# B&R Automation Studio project vibratorControlWithCurrentController
Automation Studio 4.12.5.95 SP; technology packages: Acp10Arnc0 5.23.1

## Configuration CM20

CPU X20CP0484, AutomationRuntime H4.93, Build 4.1.2, Safety 0.0, Vc 

### Task classes (Cpu.sw)
```
Cyclic#1 (cycle 800 us, tolerance 0 us):
  VibratorCo <- modules.main.vibrator.VibratorControl.prg
Cyclic#2 (cycle 1600 us, tolerance 0 us):
  sineWaveGe <- modules.main.vibrator.sineWaveGen.prg [disabled]
  belt <- modules.main.belt.belt.prg
  sampling <- modules.sampling.prg
Cyclic#3 (cycle 4800 us, tolerance 0 us):
  main <- modules.main.main.prg
  feeder <- modules.feeder.feeder.prg
  vibrator <- modules.main.vibrator.vibrator.prg
  EM_vibrat <- modules.main.vibrator.EM_Vibrator.prg
  capcon <- modules.main.capcon.capcon.prg
  wing <- modules.main.wing.wing.prg
  upperFlap <- modules.main.wing.upperFlap.upperFlap.prg
  middleFlap <- modules.main.wing.middleFlap.middleFlap.prg
  bottomFlap <- modules.main.wing.bottomFlap.bottomFlap.prg
  cassette <- modules.main.wing.cassette.cassette.prg
Cyclic#4 (cycle 20000 us, tolerance 1000000 us):
  ethIp <- services.EthernetIP.ethIp.prg
  udpClient <- services.machine.udpClient.prg
  simulation <- simulation.simulation.prg
  lampCtrl <- services.machine.lampCtrl.prg [disabled]
Cyclic#5 (cycle 40000 us, tolerance 1000000 us):
  alarm <- services.alarm.alarm.prg
  file <- services.file.file.prg
  recipe <- services.recipe.recipe.prg
  recipeCurr <- services.recipe.recipeCurrent.prg
  machine <- services.machine.machine.prg
  config <- services.config.config.prg
  updateCM <- services.machine.updateCM.prg
  updateEWU <- services.machine.updateEWU.prg
  elementImg <- services.elementImg.elementImg.prg
  simCapcon <- simulation.capcon.simCapcon.prg [disabled]
  recipeCtrl <- services.recipeCtrl.recipeCtrl.prg
  transferCo <- services.machine.transferConfigToT50.prg
  FAT <- services.FAT.FAT.prg
DataObjects: eipconf <- services.EthernetIP.eipconf.dob, Acp10sys
NcDataObjects: acp10etxen <- acp10etxen.dob, gAxisVibCi <- gAxisVibCobj.gAxisVibCi.dob, cfCurCtr <- gAxisVibCobj.cfCurCtr.dob, gAxisVibLi <- gAxisVibLobj.gAxisVibLi.dob, lfCurCtr <- gAxisVibLobj.lfCurCtr.dob, gAxisBelta <- gAxisBeltobj.gAxisBelta.dob, gAxisBelti <- gAxisBeltobj.gAxisBelti.dob, lfNew <- gAxisVibLobj.lfNew.dob
Binaries: mvLoader, udbdef, FWRules, TCData, TCLang, OpcUaSrv, arsvcreg, acp10cfg, Acp10map, arconfig, User, iomap, asfw, ashwac, ashwd, sysconf, Role, mp_recipe, mp_recipeC, asiol1, User_1, mp_config, mp_data, alarm_hist, TC, mp_user, mp_alarm
Libraries: Acp10man, Acp10par, NcGlobal, VibCtrl, LookupTbl, MpRecipe, MpBase, sys_lib, runtime, MpAlarmX, astime, brdkMC, Acp10_MC, AsBrMath, standard, AsBrStr, brsystem, brdkMU, brdkSIM, brdkCSV, brdkPV, legoCM20, legoSTR, DataObj, brdkOPCUA, AsOpcUas, brdkUpdate, ArProject, brdkFile, AsSem, AsIO, AsOpcUac, FileIO, AsIODiag, AsUSB, brdkREST, brdkJSON, brdkSTR, RandomLib, AsHttp, AsARCfg, AsMath, asstring, AsEthIP, MTFilter, MTTypes, MTBasics, MTLookUp, MTData, MpData, MpServer, Goertzel, EasyUaClnt, AsIOLink, AsIOAcc, AsUDP, powerlnk, arssl, asieccon, aruser, MpReport
```

### Hardware
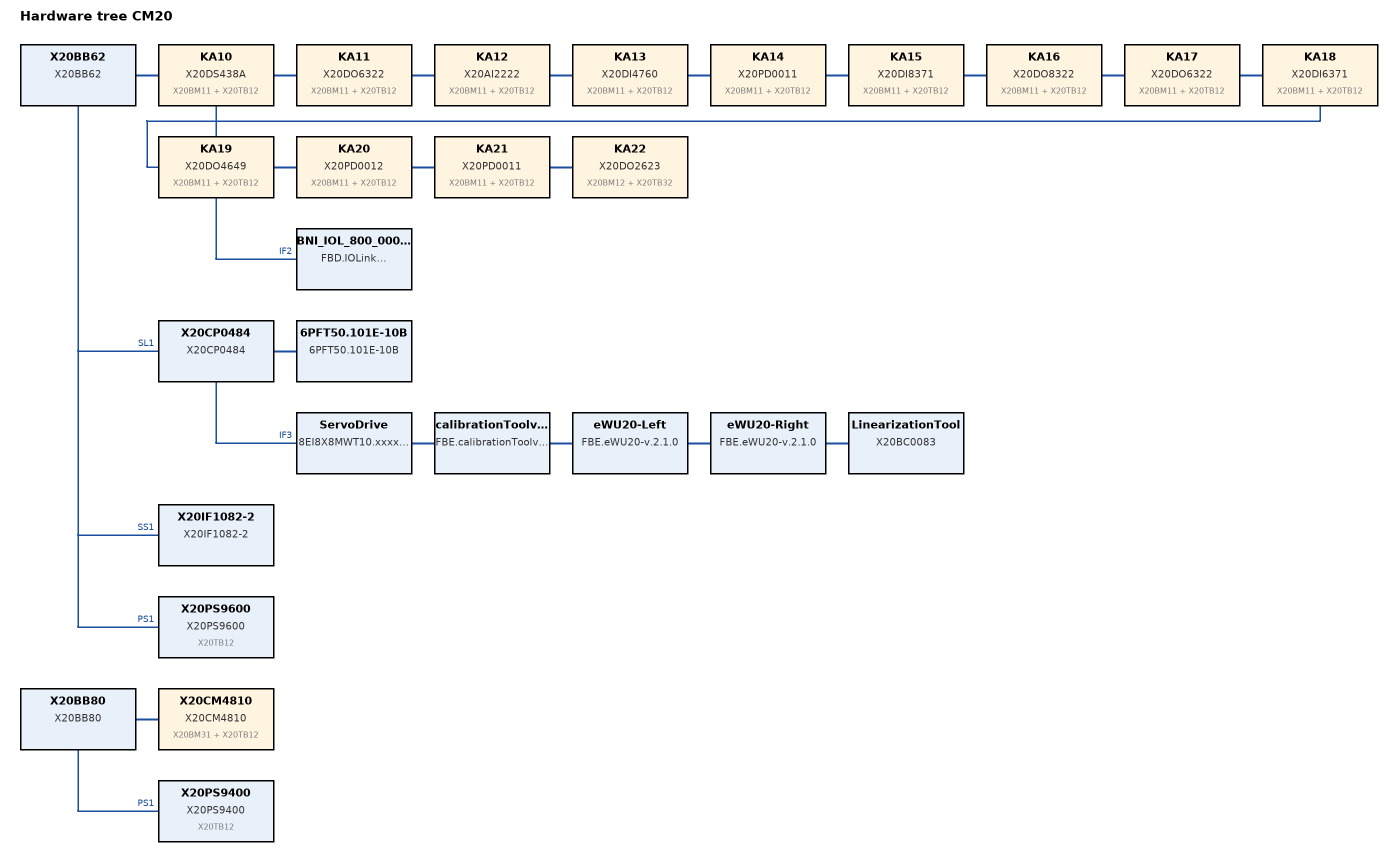
```
6PFT50.101E-10B : 6PFT50.101E-10B v1.4.0.0  [ETH1 -> X20CP0484.IF2 [Cable Type=PowerlinkCable, Length=10, Version=1.0.0.3]]
  Terminal = true
  Startmode = 2
  Mode = Manual
  InternetAddress = 192.168.2.70
  Subnetmask = 255.255.255.0
  ScreenRotation = 270
  PasswordVNC = 
  SelectedFavoriteWeb = 192.168.2.11:81
  USBmemshare = 1
  Usermemshare = 1
  PasswordCIFS = 1234
  UpdateServerType = 2
  UpdateServerFromDhcp = 0
  UpdateServerUser = superuser
  UpdateServerPassword = superuser
  UpdateServerAddress = 192.168.2.11
  PasswordService = 
  ActivateOpcUaServer = 1
BNI_IOL_800_000_Z036_IODD1_1 : FBD.IOLink.GenericDeviceDTM.DTMCore.BNI IOL-800-000-Z036 IODD1.1 v1.8 (OrderNumber=BNI IOL-800-000-Z036 IODD1.1)  [IO-Link1 -> KA10.IF2]
  DtmId = 7a61ab58-0b64-4e0b-ae65-61df76657b3c
KA10 : X20DS438A v2.4.0.0  [SS1 -> X20TB12c.SS; SL -> X20BM11b.SL1]
  DtmRef = FBD.BRIOLinkModuleDTM.DTMCore.X20DS438A
  DtmId = c2005f39-6d59-4b1f-87b2-556bc89c9aff
  CommDtmId = f866141b-695e-453b-bc4e-9ec5edcbb4a9
  RequiresDTMBuild = true
  ConfigFile = Communication.dtm
  ConfigModule = asiol1
  Supervision = off
  OperatingMode01 = DigInput
  OperatingMode02 = Operate
  PDO_Enable02 = variousTypes
  PDO_DataType02_1 = USINT
  OperatingMode03 = DigInput
KA11 : X20DO6322 v1.4.0.0  [SS1 -> X20TB12n.SS; SL -> X20BM11j.SL1]
  Supervision = off
KA12 : X20AI2222 v1.4.0.0  [SS1 -> X20TB12i.SS; SL -> X20BM11h.SL1]
  Supervision = off
KA13 : X20DI4760 v1.2.0.0  [SS1 -> X20TB12p.SS; SL -> X20BM11l.SL1]
  Supervision = off
KA14 : X20PD0011 v1.2.0.0  [SS1 -> X20TB12o.SS; SL -> X20BM11k.SL1]
  Supervision = off
KA15 : X20DI8371 v1.6.0.0  [SS1 -> X20TB12q.SS; SL -> X20BM11m.SL1]
  Supervision = off
KA16 : X20DO8322 v1.8.0.0  [SS1 -> X20TB12r.SS; SL -> X20BM11n.SL1]
  Supervision = off
KA17 : X20DO6322 v1.4.0.0  [SS1 -> X20TB12s.SS; SL -> X20BM11o.SL1]
  Supervision = off
KA18 : X20DI6371 v1.2.0.0  [SS1 -> X20TB12t.SS; SL -> X20BM11p.SL1]
  Supervision = off
KA19 : X20DO4649 v1.2.0.0  [SS1 -> X20TB12u.SS; SL -> X20BM11q.SL1]
  Supervision = off
KA20 : X20PD0012 v1.2.0.0  [SS1 -> X20TB12a.SS; SL -> X20BM11.SL1]
  Supervision = off
KA21 : X20PD0011 v1.2.0.0  [SS1 -> X20TB12b.SS; SL -> X20BM11a.SL1]
  Supervision = off
KA22 : X20DO2623 v1.2.1.0  [SS1 -> X20TB32.SS; SL -> X20BM12.SL1]
  Supervision = off
LinearizationTool : X20BC0083 v2.9.0.0  [PLK1 -> eWU20-Right.PLK2 (NodeNumber=3) [Cable Type=PowerlinkCable, Length=10, Version=1.0.0.3]; SL -> X20BB80.SL1]
  Supervision = off
ServoDrive : 8EI8X8MWT10.xxxx-1 v2.3.2.0  [PLK1 -> X20CP0484.IF3 (NodeNumber=1) [Cable Type=PowerlinkCable, Length=10, Version=1.0.0.3]; PLK2 -> calibrationToolv.1.2.0.PLK1 (NodeNumber=1) [Cable Type=PowerlinkCable, Length=10, Version=1.0.0.3]]
  MotionTP = Acp10Arnc0
  Ax1Interface = Ax1EnDat
X20BB62 : X20BB62 v1.3.0.0
  Connector IF6:
    CycleTime = 1600
    AsyncPayload = 120
    OutputJustInTime = off
X20BB80 : X20BB80 v1.0.2.0
X20BM11 : X20BM11 v1.1.0.0  [X2X1 -> X20BM11q.X2X2]
X20BM11a : X20BM11 v1.1.0.0  [X2X1 -> X20BM11.X2X2]
X20BM11b : X20BM11 v1.1.0.0  [X2X1 -> X20BB62.IF6]
X20BM11h : X20BM11 v1.1.0.0  [X2X1 -> X20BM11j.X2X2]
X20BM11j : X20BM11 v1.1.0.0  [X2X1 -> X20BM11b.X2X2]
X20BM11k : X20BM11 v1.1.0.0  [X2X1 -> X20BM11l.X2X2]
X20BM11l : X20BM11 v1.1.0.0  [X2X1 -> X20BM11h.X2X2]
X20BM11m : X20BM11 v1.1.0.0  [X2X1 -> X20BM11k.X2X2]
X20BM11n : X20BM11 v1.1.0.0  [X2X1 -> X20BM11m.X2X2]
X20BM11o : X20BM11 v1.1.0.0  [X2X1 -> X20BM11n.X2X2]
X20BM11p : X20BM11 v1.1.0.0  [X2X1 -> X20BM11o.X2X2]
X20BM11q : X20BM11 v1.1.0.0  [X2X1 -> X20BM11p.X2X2]
X20BM12 : X20BM12 v1.1.0.0  [X2X1 -> X20BM11a.X2X2]
X20BM31 : X20BM31 v1.1.0.0  [X2X1 -> X20BB80.IF1]
X20CM4810 : X20CM4810 v1.4.4.0  [SS1 -> X20TB12e.SS; SL -> X20BM31.SL1]
  Supervision = off
  AIScale01 = 0x0007
  Current02 = on
  AIScale02 = 0x0060
  AICalc02 = on
  AISamplesSource02 = cyclic
  AIParameter02 = PEAK
X20CP0484 : X20CP0484 v1.7.0.0  [SL -> X20BB62.SL1]
  Connector IF2:
    ActivateDevice = 1
    HostName = countingmachine
    Mode = Manual
    InternetAddress = 192.168.2.11
    SubnetMask = 255.255.255.0
    InaNodeNumber = 0
    ActivateSnmp = 2
  Connector IF3:
    MtuSize = 1500
    CycleTime = 800
    InternetAddress = 192.168.200.240
    SubnetMask = 255.255.255.0
    ActivateANSL = 1
  ConfigurationID = CountingMachine
  ConfigVersion = 2.1.42
  UserPartitionSize = 100
  RemanentGlobalPvSize = 500
  VolatileGlobalPvSize = 455350
  EnableUsbRemoteInstall = 1
  EnableCfRemoteInstall = 1
  TimerDeviceType = EPLX2X
  TimerDevice = X20CP0484.IF3
  IdleTaskClass = 4
  TaskClassIdleTime = 1600
  CyclicTaskClassCount = 5
  Cyclic1Duration = 800
  Cyclic1Tolerance = 0
  Cyclic2Duration = 1600
  Cyclic2Tolerance = 0
  Cyclic3Duration = 4800
  Cyclic3Tolerance = 0
  Cyclic4Duration = 20000
  Cyclic4Tolerance = 1000000
  Cyclic5Duration = 40000
  Cyclic5Tolerance = 1000000
  Cyclic6Duration = 500000
  Cyclic6Tolerance = 500000
  Cyclic7Duration = 1000000
  Cyclic7Tolerance = 1000000
  Cyclic8Duration = 9600
  Cyclic8Tolerance = 30000000
  FileDevice1
  FileDeviceName1 = USER
  FileDevicePath1 = USER_PATH
  TimeZone = 140
  ActivateSntp = 1
  SntpcServAddr1 = 192.168.1.199
  EthernetHostName = cm20
  EthernetDefaultGateway = 192.168.1.254
  ActivateDns = 1
  DnsServer1 = 192.168.1.1
  FtpUser1
  FtpUsername1 = admin
  FtpUserPassword1 = /xeWp7dP4cZARaoRUYb4lC4ZD6ydIPKFJHxZK63t4D4=
  FtpUserSalt1 = z+XtgaLv
  FTPAccessRight1 = 0
  FtpUser2
  FtpUsername2 = superuser
  FtpUserPassword2 = hun78AKmVJbSvtD9VGxdA3Iq+bPiFMAeRRsTULM9hlc=
  FtpUserSalt2 = IDYkuK0C
  FTPAccessRight2 = 0
  FTPdevice2 = ALL
  FtpUser3
  FtpUsername3 = update
  FtpUserPassword3 = +43P0CP5LPvLZS5Hk18lIwvQq9JpaLJM6nsEQnrbHXY=
  FtpUserSalt3 = TaVVG8PK
  FTPAccessRight3 = 0
  FTPMSpath3 = update
  FtpUser4
  FtpUsername4 = updateewu
  FtpUserPassword4 = epKGN9X0JvLfxgCXyMdS0yy+jyVnLXtvgYSXuK2LydA=  // updateewu
  FtpUserSalt4 = ShQX0Ew+
  FTPAccessRight4 = 0
  FTPMSpath4 = updateewu
  ActivateOpcUa = 1
  OpcUaInformationModels_PV_Version = 2
  OpcUaInformationModel_Facet = 0
  OpcUaInformationModel_TypeInformation = 0
  OpcUaInformationModel_BaseObjectTypeForStructures = 0
X20IF1082-2 : X20IF1082-2 v1.15.0.0  [SS -> X20BB62.SS1]
  Connector IF1:
    Operation = EthOnly
    HostName = cm20
    ActivateANSL = 1
    ActivateSnmp = 2
X20PS9400 : X20PS9400 v1.8.0.0  [SS1 -> X20TB12d.SS; PS -> X20BB80.PS1]
  Supervision = off
X20PS9600 : X20PS9600 v1.6.1.0  [PS -> X20BB62.PS1; SS1 -> X20TB12.SS]
X20TB12 : X20TB12 v1.0.0.0
X20TB12a : X20TB12 v1.0.0.0
X20TB12b : X20TB12 v1.0.0.0
X20TB12c : X20TB12 v1.0.0.0
X20TB12d : X20TB12 v1.0.0.0
X20TB12e : X20TB12 v1.0.0.0
X20TB12i : X20TB12 v1.0.0.0
X20TB12n : X20TB12 v1.0.0.0
X20TB12o : X20TB12 v1.0.0.0
X20TB12p : X20TB12 v1.0.0.0
X20TB12q : X20TB12 v1.0.0.0
X20TB12r : X20TB12 v1.0.0.0
X20TB12s : X20TB12 v1.0.0.0
X20TB12t : X20TB12 v1.0.0.0
X20TB12u : X20TB12 v1.0.0.0
X20TB32 : X20TB32 v1.0.0.1
calibrationToolv.1.2.0 : FBE.calibrationToolv.1.2.0 v1.0 (OrderNumber=calibrationToolv.1.2.0)  [PLK1 -> ServoDrive.PLK2 (NodeNumber=2) [Cable Type=PowerlinkCable, Length=10, Version=1.0.0.3]; PLK2 -> eWU20-Left.PLK1 (NodeNumber=2) [Cable Type=PowerlinkCable, Length=10, Version=1.0.0.3]]
  Supervision = off
  pA240s01_direction = ro
  pA240s03_direction = ro
  pA500s01_direction = wo
eWU20-Left : FBE.eWU20-v.2.1.0 v1.0 (OrderNumber=eWU20-Left)  [PLK1 -> calibrationToolv.1.2.0.PLK2 (NodeNumber=20) [Cable Type=PowerlinkCable, Length=10, Version=1.0.0.3]; PLK2 -> eWU20-Right.PLK1 (NodeNumber=20) [Cable Type=PowerlinkCable, Length=10, Version=1.0.0.3]]
  Supervision = off
  pA080s01_direction = ro
  pA080s02_direction = ro
  pA080s03_direction = ro
  pA080s04_direction = ro
  pA080s05_direction = ro
  pA080s06_direction = ro
  pA080s07_direction = ro
  pA080s08_direction = ro
  pA080s09_direction = ro
  pA080s0A_direction = ro
  pA080s0B_direction = ro
  pA500s01_direction = wo
  pA500s02_direction = wo
  pA500s03_direction = wo
  pA500s04_direction = wo
  pA500s05_direction = wo
  pA500s06_direction = wo
  pA500s07_direction = wo
  pA500s08_direction = wo
  pA500s09_direction = wo
  pA500s0A_direction = wo
  pA500s0B_direction = wo
  pA500s0C_direction = wo
  pA500s0D_direction = wo
  pA500s0E_direction = wo
  pA1C0s01_direction = ro
  pA1C0s02_direction = ro
  pA1C0s03_direction = ro
  pA1C0s04_direction = ro
eWU20-Right : FBE.eWU20-v.2.1.0 v1.0 (OrderNumber=eWU20-Left)  [PLK1 -> eWU20-Left.PLK2 (NodeNumber=21) [Cable Type=PowerlinkCable, Length=10, Version=1.0.0.3]; PLK2 -> LinearizationTool.PLK1 (NodeNumber=21) [Cable Type=PowerlinkCable, Length=10, Version=1.0.0.3]]
  Supervision = off
  pA080s01_direction = ro
  pA080s02_direction = ro
  pA080s03_direction = ro
  pA080s04_direction = ro
  pA080s05_direction = ro
  pA080s06_direction = ro
  pA080s07_direction = ro
  pA080s08_direction = ro
  pA080s09_direction = ro
  pA080s0A_direction = ro
  pA080s0B_direction = ro
  pA500s01_direction = wo
  pA500s02_direction = wo
  pA500s03_direction = wo
  pA500s04_direction = wo
  pA500s05_direction = wo
  pA500s06_direction = wo
  pA500s07_direction = wo
  pA500s08_direction = wo
  pA500s09_direction = wo
  pA500s0A_direction = wo
  pA500s0B_direction = wo
  pA500s0C_direction = wo
  pA500s0D_direction = wo
  pA500s0E_direction = wo
  pA1C0s01_direction = ro
  pA1C0s02_direction = ro
  pA1C0s03_direction = ro
  pA1C0s04_direction = ro
```

### Cpu.pkg.orig - X20CP0484/Cpu.pkg.orig
(orig body not rendered)

### IoMap.iom - X20CP0484/IoMap.iom
```iecst
VAR_CONFIG
	::feeder:this.hw.do_levelSensorInBowlLow AT %QX."KA11".DigitalOutput01;
	::feeder:this.hw.do_levelSensorInBowlMedium AT %QX."KA11".DigitalOutput03;
	::feeder:this.hw.do_levelSensorInBowlHigh AT %QX."KA11".DigitalOutput05;
	::main:this.hw.do_alarmBeacon AT %QX."KA11".DigitalOutput02;
	::main:this.alarm.KA11.active AT %IX."KA11".ModuleOk;
	::feeder:this.hw.do_beltForwards AT %QX."KA11".DigitalOutput04;
	::feeder:this.hw.do_beltBackwards AT %QX."KA11".DigitalOutput06;
	::main:this.alarm.KA12.active AT %IX."KA12".ModuleOk;
	::sampling:this.hw.ai_signal[1] AT %IW."KA12".AnalogInput01;
	::sampling:this.hw.di_upperFlap_change AT %IX."KA13".DigitalInput01;
	::sampling:this.hw.di_bottomFlap_change AT %IX."KA13".DigitalInput02;
	::sampling:this.hw.di_middleFlap_change AT %IX."KA13".DigitalInput03;
	::sampling:this.hw.di_neigbourFlap_change AT %IX."KA13".DigitalInput04;
	::main:this.alarm.KA14.active AT %IX."KA13".ModuleOk;
	::main:this.alarm.KA13.active AT %IX."KA14".ModuleOk;
	::cassette:this.hwAir.di_neighbourActive AT %IX."KA15".DigitalInput02;
	::cassette:this.hwAir.di_cassetteReady AT %IX."KA15".DigitalInput03;
	::bottomFlap:this.hwAir.di_neighbourPortionReady AT %IX."KA15".DigitalInput05;
	::cassette:this.hwAir.di_cassetteQueue AT %IX."KA15".DigitalInput01;
	::bottomFlap:this.hwAir.di_neighbourActive AT %IX."KA15".DigitalInput02;
	::cassette:this.hwAir.di_neighbourIsDosing AT %IX."KA15".DigitalInput04;
	::cassette:this.hwAir.di_neighbourBricksInCassette AT %IX."KA15".DigitalInput07;
	::main:this.alarm.KA15.active AT %IX."KA15".ModuleOk;
	::bottomFlap:this.hwAir.di_neigbourIsDosing AT %IX."KA15".DigitalInput04;
	::upperFlap:this.hw.do_open AT %QX."KA16".DigitalOutput01;
	::middleFlap:this.hw.do_open AT %QX."KA16".DigitalOutput03;
	::bottomFlap:this.hw.do_neighbourPortionReady AT %QX."KA16".DigitalOutput05;
	::cassette:this.hw.do_bricksReadyInCassette AT %QX."KA16".DigitalOutput07;
	::cassette:this.hw.do_dosing AT %QX."KA16".DigitalOutput04;
	::wing:this.hw.do_active AT %QX."KA16".DigitalOutput02;
	::main:this.alarm.KA16.active AT %IX."KA16".ModuleOk;
	::feeder:this.hw.do_beltForwards AT %QX."KA16".DigitalOutput06;
	::feeder:this.hw.do_beltBackwards AT %QX."KA16".DigitalOutput08;
	::bottomFlap:this.hw.do_open AT %QX."KA17".DigitalOutput01;
	::bottomFlap:this.hw.do_neighbourOpen AT %QX."KA17".DigitalOutput03;
	::cassette:this.hw.do_cassetteRelease AT %QX."KA17".DigitalOutput05;
	::main:this.alarm.KA17.active AT %IX."KA17".ModuleOk;
	::feeder:this.hw.di_flapIsClosed AT %IX."KA18".DigitalInput02;
	::feeder:this.hw.di_levelSensorBelt AT %IX."KA18".DigitalInput03;
	::feeder:this.hw.di_flapIsOpen AT %IX."KA18".DigitalInput04;
	::feeder:this.hw.di_boxIsReadyAtFlap AT %IX."KA18".DigitalInput05;
	::main:this.alarm.KA18.active AT %IX."KA18".ModuleOk;
	::feeder:this.hw.do_flapClose AT %QX."KA19".DigitalOutput01;
	::feeder:this.hw.do_flapClose AT %QX."KA19".DigitalOutput04;
	::feeder:this.hw.do_flapOpen AT %QX."KA19".DigitalOutput02;
	::feeder:this.hw.do_flapOpen AT %QX."KA19".DigitalOutput03;
	::main:this.alarm.KA19.active AT %IX."KA19".ModuleOk;
	::main:this.alarm.KA20.active AT %IX."KA20".ModuleOk;
	::main:this.alarm.KA21.active AT %IX."KA21".ModuleOk;
	::main:this.alarm.KA10.active AT %IX."KA10".ModuleOk;
	::feeder:this.hw.di_levelSensorInBowl AT %IX."KA10".DigitalInput01;
	::belt:this.hw.di_photo AT %IX."KA10".DigitalInput03;
	::VibratorCo:localVariables[1].Accelerometer_0.ai_peakValue AT %ID."calibrationToolv.1.2.0".AnalogValue_IA240_S01;
	::VibratorCo:localVariables[1].Accelerometer_0.ai_rawValue AT %ID."calibrationToolv.1.2.0".RawVib_IA240_S03;
	::VibratorCo:localVariables[0].Accelerometer_0.ai_rawValue AT %ID."calibrationToolv.1.2.0".RawVib_IA240_S03;
	::sineWaveGe:acc.analogVib AT %ID."calibrationToolv.1.2.0".AnalogValue_IA240_S01;
	::VibratorCo:localVariables[0].Accelerometer_0.ai_peakValue AT %ID."calibrationToolv.1.2.0".AnalogValue_IA240_S01;
	::EM_vibrat:localVariables[0].hw.ModuleOkCalibrationTool AT %IX."calibrationToolv.1.2.0".ModuleOk;
	::EM_vibrat:localVariables[1].hw.ModuleOkCalibrationTool AT %IX."calibrationToolv.1.2.0".ModuleOk;
	::VibratorCo:localVariables[0].Accelerometer_0.ModuleOkCalibrationTool AT %IX."calibrationToolv.1.2.0".ModuleOk;
	::VibratorCo:localVariables[1].Accelerometer_0.ModuleOkCalibrationTool AT %IX."calibrationToolv.1.2.0".ModuleOk;
	::cassette:this.hwWu[1].di_wingUnitActive AT %IX."eWU20-Right".WuConnected_IA080_S01;
	::bottomFlap:this.hwWu[1].neighbourActive AT %IX."eWU20-Right".StatusNeighbourActive_IA080_S02;
	::cassette:this.hwWu[0].di_wingUnitActive AT %IX."eWU20-Left".WuConnected_IA080_S01;
	::upperFlap:this.hwWu[0].di_wingUnitActive AT %IX."eWU20-Left".WuConnected_IA080_S01;
	::middleFlap:this.hwWu[0].di_wingUnitActive AT %IX."eWU20-Left".WuConnected_IA080_S01;
	::bottomFlap:this.hwWu[0].di_wingUnitActive AT %IX."eWU20-Left".WuConnected_IA080_S01;
	::bottomFlap:this.hwWu[0].neighbourActive AT %IX."eWU20-Left".StatusNeighbourActive_IA080_S02;
	::bottomFlap:this.hwWu[0].neigbourIsDosing AT %IX."eWU20-Left".Di_bottomFlap_neighbourIsDosing_IA080_S03;
	::bottomFlap:this.hwWu[0].neighbourPortionReady AT %IX."eWU20-Left".Di_bottomFlap_neighbourPortReady_IA080_S04;
	::cassette:this.hwWu[0].di_cassetteQueue AT %IX."eWU20-Left".Di_cassette_queue_IA080_S05;
	::cassette:this.hwWu[0].di_neighbourActive AT %IX."eWU20-Left".Di_cassette_neighbourActive_IA080_S06;
	::cassette:this.hwWu[0].di_cassetteReady AT %IX."eWU20-Left".Di_cassette_ready_IA080_S07;
	::cassette:this.hwWu[0].di_neighbourIsDosing AT %IX."eWU20-Left".Di_cassette_neighbourIsDosing_IA080_S08;
	::cassette:this.hwWu[0].di_neighbourBricksInCassette AT %IX."eWU20-Left".Di_cassette_neighbourBricksInCas_IA080_S09;
	::bottomFlap:cm20Connected AT %QX."eWU20-Left".CM20connected_IA500_S01;
	::upperFlap:this.flap.do_open AT %QX."eWU20-Left".Do_upperFlap_open_IA500_S02;
	::middleFlap:this.flap.do_open AT %QX."eWU20-Left".Do_middleFlap_open_IA500_S03;
	::bottomFlap:this.flap.do_open AT %QX."eWU20-Left".Do_bottomFlap_open_IA500_S04;
	::bottomFlap:this.hw.do_neighbourPortionReady AT %QX."eWU20-Left".Do_bottomFlap_neighbourPortReady_IA500_S06;
	::bottomFlap:this.neighbourFlap.do_open AT %QX."eWU20-Left".Do_bottomFlap_neighbourOpen_IA500_S07;
	::cassette:this.hwWu[0].do_active AT %QX."eWU20-Left".Do_cm_active_IA500_S09;
	::cassette:this.hw.do_bricksReadyInCassette AT %QX."eWU20-Left".Do_cassette_BricksReadyInCasette_IA500_S0A;
	::cassette:this.hw.do_cassetteRelease AT %QX."eWU20-Left".Do_cassette_cassetteRelease_IA500_S0B;
	::upperFlap:this.hwWu[0].flapPosition AT %ID."eWU20-Left".Di_upperFlap_positionStatus_IA1C0_S01;
	::middleFlap:this.hwWu[0].flapPosition AT %ID."eWU20-Left".Di_middleFlap_positionStatus_IA1C0_S02;
	::bottomFlap:this.hwWu[0].flapPosition AT %ID."eWU20-Left".Di_bottomFlap_positionStatus_IA1C0_S03;
	::bottomFlap:this.hwWu[0].neighbourFlapPosition AT %ID."eWU20-Left".Di_neighbourFlap_positionStatus_IA1C0_S04;
	::upperFlap:this.hwWu[1].di_wingUnitActive AT %IX."eWU20-Right".WuConnected_IA080_S01;
	::middleFlap:this.hwWu[1].di_wingUnitActive AT %IX."eWU20-Right".WuConnected_IA080_S01;
	::bottomFlap:this.hwWu[1].di_wingUnitActive AT %IX."eWU20-Right".WuConnected_IA080_S01;
	::bottomFlap:this.hwWu[1].neigbourIsDosing AT %IX."eWU20-Right".Di_bottomFlap_neighbourIsDosing_IA080_S03;
	::bottomFlap:this.hwWu[1].neighbourPortionReady AT %IX."eWU20-Right".Di_bottomFlap_neighbourPortReady_IA080_S04;
	::cassette:this.hwWu[1].di_cassetteQueue AT %IX."eWU20-Right".Di_cassette_queue_IA080_S05;
	::cassette:this.hwWu[1].di_neighbourActive AT %IX."eWU20-Right".Di_cassette_neighbourActive_IA080_S06;
	::cassette:this.hwWu[1].di_cassetteReady AT %IX."eWU20-Right".Di_cassette_ready_IA080_S07;
	::cassette:this.hwWu[1].di_neighbourIsDosing AT %IX."eWU20-Right".Di_cassette_neighbourIsDosing_IA080_S08;
	::cassette:this.hwWu[1].di_neighbourBricksInCassette AT %IX."eWU20-Right".Di_cassette_neighbourBricksInCas_IA080_S09;
	::bottomFlap:cm20Connected AT %QX."eWU20-Right".CM20connected_IA500_S01;
	::upperFlap:this.flap.do_open AT %QX."eWU20-Right".Do_upperFlap_open_IA500_S02;
	::middleFlap:this.flap.do_open AT %QX."eWU20-Right".Do_middleFlap_open_IA500_S03;
	::bottomFlap:this.flap.do_open AT %QX."eWU20-Right".Do_bottomFlap_open_IA500_S04;
	::bottomFlap:this.hw.do_neighbourPortionReady AT %QX."eWU20-Right".Do_bottomFlap_neighbourPortReady_IA500_S06;
	::bottomFlap:this.neighbourFlap.do_open AT %QX."eWU20-Right".Do_bottomFlap_neighbourOpen_IA500_S07;
	::cassette:this.hwWu[1].do_active AT %QX."eWU20-Right".Do_cm_active_IA500_S09;
	::cassette:this.hw.do_bricksReadyInCassette AT %QX."eWU20-Right".Do_cassette_BricksReadyInCasette_IA500_S0A;
	::cassette:this.hw.do_cassetteRelease AT %QX."eWU20-Right".Do_cassette_cassetteRelease_IA500_S0B;
	::upperFlap:this.hwWu[1].flapPosition AT %ID."eWU20-Right".Di_upperFlap_positionStatus_IA1C0_S01;
	::middleFlap:this.hwWu[1].flapPosition AT %ID."eWU20-Right".Di_middleFlap_positionStatus_IA1C0_S02;
	::bottomFlap:this.hwWu[1].flapPosition AT %ID."eWU20-Right".Di_bottomFlap_positionStatus_IA1C0_S03;
	::bottomFlap:this.hwWu[1].neighbourFlapPosition AT %ID."eWU20-Right".Di_neighbourFlap_positionStatus_IA1C0_S04;
	::wing:this.hw.wu_error[0] AT %IX."eWU20-Left".Wu_error_IA080_S0A;
	::wing:this.hw.wu_error[1] AT %IX."eWU20-Right".Wu_error_IA080_S0A;
	::main:this.hw.do_wo_ON AT %QX."eWU20-Left".Di_CMRunning_IA500_S0C;
	::main:this.hw.do_wo_ON AT %QX."eWU20-Right".Di_CMRunning_IA500_S0C;
	::main:this.hw.do_clearWU AT %QX."eWU20-Left".Do_clearWU_IA500_S0D;
	::main:this.hw.do_clearWU AT %QX."eWU20-Right".Do_clearWU_IA500_S0D;
	::machine:this.warmRestartWU AT %QX."eWU20-Left".Do_warmRestartWU_IA500_S0E;
	::machine:this.warmRestartWU AT %QX."eWU20-Right".Do_warmRestartWU_IA500_S0E;
	::cassette:this.hw.do_dosing AT %QX."eWU20-Left".Do_bottomFlap_dosing_IA500_S05;
	::cassette:this.hw.do_dosing AT %QX."eWU20-Right".Do_bottomFlap_dosing_IA500_S05;
	::main:this.hw.di_stepperWUExecute[0] AT %IX."eWU20-Left".Di_WU_execute_IA080_S0B;
	::main:this.hw.di_stepperWUExecute[1] AT %IX."eWU20-Right".Di_WU_execute_IA080_S0B;
	::main:this.hw.output_lightTowerBalluff AT %QB."KA10".OutputData02_1;
	::VibratorCo:localVariables[0].Accelerometer_0.isBigCF AT %QX."calibrationToolv.1.2.0".IsBigCF_IA500_S01;
	::VibratorCo:localVariables[1].Accelerometer_0.ai_peakValueBusCtrl AT %ID."X20CM4810".AnalogInput02;
	Cyclic#1.::VibratorCo:localVariables[0].Accelerometer_0.ai_peakValueBusCtrl AT %ID."X20CM4810".AnalogInput02;
	::VibratorCo:localVariables[0].Accelerometer_0.do_enableSampling AT %QX."X20CM4810".AnalogInputControl02;
	::VibratorCo:localVariables[0].Accelerometer_0.ao_samples AT %QW."X20CM4810".AnalogInputSamples02;
	::VibratorCo:localVariables[1].Accelerometer_0.ai_rawValueBusCtrl AT %ID."X20CM4810".AnalogInput01;
	::VibratorCo:localVariables[0].Accelerometer_0.ai_rawValueBusCtrl AT %ID."X20CM4810".AnalogInput01;
	::VibratorCo:localVariables[0].Accelerometer_0.ModuleOkBusCtrl AT %IX."X20CM4810".ModuleOk;
	::VibratorCo:localVariables[1].Accelerometer_0.ModuleOkBusCtrl AT %IX."X20CM4810".ModuleOk;
	::EM_vibrat:localVariables[1].hw.ModuleOkCalibrationToolBusCtrl AT %IX."X20CM4810".ModuleOk;
	::EM_vibrat:localVariables[0].hw.ModuleOkCalibrationToolBusCtrl AT %IX."X20CM4810".ModuleOk;
	::main:this.hw.input_lightTowerBalluff AT %IB."KA10".ChannelStatus02;
END_VAR
```

### Acp10cfg.ncc - X20CP0484/Motion/Acp10cfg.ncc
```
NcConfiguration (Version=5.12.2, NcSwId=Acp10)
  ACP10CF1_typ:
    cnt_nettrc_rec_drive = 1500
    bufsize_trace_upload = 1200
    tc_nc_man_task = Cyclic #2
    glob_pv_as_ncobject = Yes
    ncsys_dl_broadcast = Yes
    ncsys_dl_acp_reset = Yes
    safemc_log_err_to_ax = Yes
    network_init:
      ncsw_init_execute = Yes
      automatic_execute = Yes
      node_nr_warning = Yes
      net_err_before_ncact = Yes
    nettrc:
      enter_parsecrec = Yes
      enter_ncaction = Yes
      save_ring_startidx = Yes
    cam_prof_download:
      cam_dat_dl_parallel = No
      tc_cam_dl_parallel = Task class for NC Manager task
    plk_if[0]:
      if_name = IF3
      tc_CycDat_PLCopen = Cyclic #1
      mc_broadcast_extdat = No
    plk_if[1]:
      if_name = IF1
      tc_CycDat_PLCopen = Task class for NC Manager task
      mc_broadcast_extdat = No
```

### Acp10map.ncm - X20CP0484/Motion/Acp10map.ncm
```
NcMapping (NcSwId=Acp10, DisabledNodesAreHidden=False)
  NcObject gAxisBelt (ModuleId=ServoDrive, Type=ncAXIS, Channel=1, AcoposSimulation=Off, InitParameter=gAxisBelti, AcoposParameter=gAxisBelta, Disabled=FALSE, ModuleDisabled=FALSE)
  NcObject gAxisVibL (ModuleId=ServoDrive, Type=ncAXIS, Channel=2, AcoposSimulation=Off, InitParameter=gAxisVibLi, AcoposParameter=lfNew, Disabled=FALSE, ModuleDisabled=FALSE)
  NcObject 8EI8X8MWT10.xxxx-1_ncV_AXIS1 (ModuleId=ServoDrive, Type=ncV_AXIS, Channel=1, Disabled=TRUE, ModuleDisabled=FALSE)
  NcObject 8EI8X8MWT10.xxxx-1_ncV_AXIS2 (ModuleId=ServoDrive, Type=ncV_AXIS, Channel=2, Disabled=TRUE, ModuleDisabled=FALSE)
  NcObject gAxisVibC (ModuleId=ServoDrive, Type=ncAXIS, Channel=3, AcoposSimulation=Off, InitParameter=gAxisVibCi, AcoposParameter=cfCurCtr, Disabled=FALSE, ModuleDisabled=FALSE)
  NcObject ServoDrive_ncV_AXIS3 (ModuleId=ServoDrive, Type=ncV_AXIS, Channel=3, AcoposSimulation=off, Disabled=true, ModuleDisabled=FALSE)
```

### beltCapcon.vvm - X20CP0484/beltCapcon.vvm
```iecst
(*Belt --> Capcon*)
(*Capcon --> Belt*)
VAR_CONFIG
	Cyclic#3.gCapconInterface.status.ready AT %Q.Cyclic#2.gBeltInterface.cmd.dropBrick; (*Command to belt that the capcon is ready for a brick*)
	Cyclic#3.::gCapconInterface.status.numBricksInPortion AT %Q.Cyclic#2.::gBeltInterface.parameter.brickCountInPortion; (*Insert your comment here...*)
END_VAR
```

### beltFeeder.vvm - X20CP0484/beltFeeder.vvm
```iecst
(*Belt --> Feeder*)
VAR_CONFIG
	Cyclic#2.::gBeltInterface.status.speed AT %Q.Cyclic#3.::gFeederInterface.cmd.speed; (*Insert your comment here...*)
END_VAR
```

### capconWing.vvm - X20CP0484/capconWing.vvm
```iecst
VAR_CONFIG
	Cyclic#3.gWingInterface.status.request AT %Q.Cyclic#3.gCapconInterface.cmd.wingRequest; (*Insert your comment here...*)
	Cyclic#3.gWingInterface.status.ready AT %Q.Cyclic#3.gCapconInterface.cmd.wingReady; (*Insert your comment here...*)
	Cyclic#3.::gCapconInterface.status.wingStartBrickNOK AT %Q.Cyclic#3.::gWingInterface.cmd.startBrickNOK; (*Start wing with brick NOK.*)
	Cyclic#3.::gCapconInterface.status.wingStartBrickOK AT %Q.Cyclic#3.::gWingInterface.cmd.startBrickOK; (*Start wing with brick OK.*)
	Cyclic#3.::gCapconInterface.status.wingStart AT %Q.Cyclic#3.::gWingInterface.cmd.startBrick; (*Start wing without status yet*)
	Cyclic#3.::gWingInterface.status.commandAck AT %Q.Cyclic#3.gCapconInterface.cmd.wingCmdAck; (*Insert your comment here...*)
	Cyclic#3.::gCapconInterface.status.wingDosing AT %Q.Cyclic#3.::gCassetteInterface.cmd.dosing; (*Insert your comment here...*)
END_VAR
```

### mainBelt.vvm - X20CP0484/mainBelt.vvm
```iecst
(*Main --> Belt*)
VAR_CONFIG
	Cyclic#3.::gMainInterface.status.doCalibrate AT %Q.Cyclic#3.::gBeltInterface.cmd.calibrate; (*Insert your comment here...*)
END_VAR
(*Belt --> Main*)
VAR_CONFIG
	Cyclic#3.::gBeltInterface.status.calibratingMode AT %Q.Cyclic#3.::gMainInterface.cmd.activateCalibrateMode[0]; (*Insert your comment here...*)
END_VAR
```

### mainCapcon.vvm - X20CP0484/mainCapcon.vvm
```iecst
(*Main --> Capcon*)
VAR_CONFIG
	Cyclic#3.::gMainInterface.status.doCalibrate AT %Q.Cyclic#3.::gCapconInterface.cmd.emptyStop; (*Insert your comment here...*)
	Cyclic#3.::gMainInterface.status.emptying AT %Q.Cyclic#3.::gCapconInterface.cmd.skipTeach; (*Insert your comment here...*)
END_VAR
(*Capon --> Main*)
VAR_CONFIG
	Cyclic#3.gCapconInterface.status.waiting AT %Q.Cyclic#3.::gMainInterface.cmd.capconWaiting; (*Command to belt that the capcon is ready for a brick*)
END_VAR
```

### mainFeeder.vvm - X20CP0484/mainFeeder.vvm
```iecst
(*Main --> Feeder*)
VAR_CONFIG
	Cyclic#3.::gMainInterface.status.feederStart AT %Q.Cyclic#3.::gFeederInterface.cmd.start; (*Insert your comment here...*)
	Cyclic#3.::gMainInterface.status.feederStop AT %Q.Cyclic#3.::gFeederInterface.cmd.stop; (*Insert your comment here...*)
END_VAR
```

### mainToWing.vvm - X20CP0484/mainToWing.vvm
```iecst
(*Main --> Wing*)
VAR_CONFIG
	Cyclic#3.::gMainInterface.line.emptyMode AT %Q.Cyclic#3.::gWingInterface.cmd.shaftModeEmpty; (*Insert your comment here...*)
	Cyclic#3.::gBottomFlapInterface.status.ready1 AT %Q.Cyclic#3.::gMainInterface.cmd.wingReadyToEmpty; (*Insert your comment here...*)
END_VAR
```

### mainVibr.vvm - X20CP0484/mainVibr.vvm
```iecst
(*Main --> vibrators*)
VAR_CONFIG
	Cyclic#3.::gMainInterface.status.doCalibrate AT %Q.Cyclic#3.::gVibratorInterface[0].cmd.calibrate; (*Insert your comment here...*)
	Cyclic#3.::gMainInterface.status.doCalibrate AT %Q.Cyclic#3.::gVibratorInterface[1].cmd.calibrate; (*Insert your comment here...*)
END_VAR
(*Vibrators --> main*)
VAR_CONFIG
	Cyclic#3.::gVibratorInterface[1].status.calibratingMode AT %Q.Cyclic#3.::gMainInterface.cmd.activateCalibrateMode[2]; (*Insert your comment here...*)
	Cyclic#3.::gVibratorInterface[0].status.calibratingMode AT %Q.Cyclic#3.::gMainInterface.cmd.activateCalibrateMode[1]; (*Insert your comment here...*)
END_VAR
```

### alarm_hist.mpalarmxhistory - X20CP0484/mappServices/alarm_hist.mpalarmxhistory
```
Element mpAlarmXHistory (Type=mpalarmxhistory)
```

### mp_alarm.mpalarmxcore - X20CP0484/mappServices/mp_alarm.mpalarmxcore
```
Element mpAlarmXCore (Type=mpalarmxcore)
  mapp.AlarmX.Core:
    BySeverity:
      [0]:
        Severity = 1  // severity 1 abort Main
        [0] = Reaction
          Name = abortMain
        [1] = Reaction
          Name = alarmBeaconFlash
      [1]:
        Severity = 10  // Severity 10 is abort  Feeder
        [0] = Reaction
          Name = alarmBeaconFlash
        [1] = Reaction
          Name = abortFeeder
      [2]:
        Severity = 20  // Severity 20 is abort CF
        [0] = Reaction
          Name = abortMain
        [1] = Reaction
          Name = alarmBeaconFlash
        [2] = Reaction
          Name = abortCircularFeeder
      [3]:
        Severity = 30  // Severity 30 is abort LF
        [0] = Reaction
          Name = abortMain
        [1] = Reaction
          Name = alarmBeaconFlash
        [2] = Reaction
          Name = abortLinearFeeder
      [4]:
        Severity = 40  // Severity 40 is abort Belt
        [0] = Reaction
          Name = abortMain
        [1] = Reaction
          Name = alarmBeaconFlash
        [2] = Reaction
          Name = abortBelt
      [5]:
        Severity = 50  // Severity 50 is abort Capcon
        [0] = Reaction
          Name = abortMain
        [1] = Reaction
          Name = alarmBeaconFlash
        [2] = Reaction
          Name = abortCapcon
      [6]:
        Severity = 60  // Severity 60 is abort Wing
        [0] = Reaction
          Name = abortWing
        [1] = Reaction
          Name = alarmBeaconFlash
        [2] = Reaction
          Name = abortMain
      [7]:
        Severity = 70
        [0] = Reaction
          Name = abortMain
        [1] = Reaction
          Name = abortFeeder
      [8]:
        Severity = 1000  // Severity 1000 is a warning - will show constant light on alarm beacon
        [0] = Reaction
          Name = alarmBeaconOn
      [9]:
        Severity = 1001  // Severity 1001 is a warning - will blink the alarm beacon slow.
        [0] = Reaction
          Name = alarmBeaconFlashSlow
  mapp.AlarmX.Core.Configuration:
    [0]:
      Name = KA10ModuleError
      Message = {$MainAlarms/KA10ModuleError}
      Code = 100
    [1]:
      Name = KA11ModuleError
      Message = {$MainAlarms/KA11ModuleError}
      Code = 101
    [2]:
      Name = KA12ModuleError
      Message = {$MainAlarms/KA12ModuleError}
      Code = 102
    [3]:
      Name = KA13ModuleError
      Message = {$MainAlarms/KA13ModuleError}
      Code = 103
    [4]:
      Name = KA14ModuleError
      Message = {$MainAlarms/KA14ModuleError}
      Code = 104
    [5]:
      Name = KA15ModuleError
      Message = {$MainAlarms/KA15ModuleError
      Code = 105
    [6]:
      Name = KA16ModuleError
      Message = {$MainAlarms/KA16ModuleError}
      Code = 106
    [7]:
      Name = KA17ModuleError
      Message = {$MainAlarms/KA17ModuleError}
      Code = 107
    [8]:
      Name = KA18ModuleError
      Message = {$MainAlarms/KA18ModuleError}
      Code = 108
    [9]:
      Name = KA19ModuleError
      Message = {$MainAlarms/KA19ModuleError}
      Code = 109
    [10]:
      Name = KA20ModuleError
      Message = {$MainAlarms/KA20ModuleErrorr}
      Code = 110
    [11]:
      Name = feederLowLevel
      Message = {$FeederAlarms/lowLevel}
      Code = 200
      Severity = 1000
    [12]:
      Name = feederBoxMissing
      Message = {$FeederAlarms/boxMissing}
      Code = 201
      Severity = 1000
    [13]:
      Name = feederCannotCloseFlap
      Message = {$FeederAlarms/cannotCloseFlap}
      Code = 202
      Severity = 10
    [14]:
      Name = feederCannotOpenFlap
      Message = {$FeederAlarms/cannotOpenFlap}
      Code = 203
      Severity = 70  // abort both main and feeder
    [15]:
      Name = circularFeederAxisFault
      Message = {&circularFeederFaultText}
      Code = 300
      Severity = 20
    [16]:
      Name = linearFeederAxisFault
      Message = {&linearFeederFaultText}
      Code = 400
      Severity = 30
    [17]:
      Name = beltMissingElements
      Message = {$BeltAlarms/missingElements}
      Code = 506
      Severity = 1001
    [18]:
      Name = beltAxisError
      Message = {$BeltAlarms/axisError}
      Code = 507
      Severity = 40
    [19]:
      Name = beltBlocked
      Message = {$BeltAlarms/beltBlocked}
      Code = 508
      Severity = 40
    [20]:
      Name = capconTeachingError
      Message = {$CapconAlarms/teachingError}
      Code = 600
      Severity = 50
    [21]:
      Name = capconOffsetError
      Message = {$CapconAlarms/offsetError}
      Code = 601
      Severity = 50
    [22]:
      Name = capconNoise
      Message = {$CapconAlarms/noise}
      Code = 602
      Severity = 50
    [23]:
      Name = upperFlapOpenTooLong
      Message = {$UpperFlapAlarms/upperFlapOpenTooLong}
      Code = 700
    [24]:
      Name = upperFlapCloseTooLong
      Message = {$UpperFlapAlarms/upperFlapCloseTooLong}
      Code = 701
    [25]:
      Name = middleFlapOpenTooLong
      Message = {$MiddleFlapAlarms/middleFlapOpenTooLong}
      Code = 800
    [26]:
      Name = middleFlapCloseTooLong
      Message = {$MiddleFlapAlarms/middleFlapCloseTooLong}
      Code = 801
    [27]:
      Name = bottomFlapOpenTooLong
      Message = {$BottomFlapAlarms/bottomFlapOpenTooLong}
      Code = 900
    [28]:
      Name = bottomFlapCloseTooLong
      Message = {$BottomFlapAlarms/bottomFlapCloseTooLong}
      Code = 901
    [29]:
      Name = neighbourBottomFlapOpenTooLong
      Message = {$BottomFlapAlarms/bottomNeighbourOpenTooLong}
      Code = 902
    [30]:
      Name = neighbourBottomFlapCloseTooLong
      Message = {$BottomFlapAlarms/bottomNeighbourCloseTooLong}
      Code = 903
    [31]:
      Name = neighbourNotActive
      Message = {$BottomFlapAlarms/neighbourNotActive}
      Code = 904
    [32]:
      Name = offsetErrorCurrent
      Code = 37
    [33]:
      Name = offsetErrorVoltage
      Code = 38
    [34]:
      Name = CMerrorHigh
      Code = 39
    [35]:
      Name = modulationOffset
      Code = 41
    [36]:
      Name = phaseRegulation
      Code = 42
    [37]:
      Name = noCoreSaturation
      Code = 43
    [38]:
      Name = brakeError
      Code = 44
    [39]:
      Name = powerCircuitError
      Code = 45
    [40]:
      Name = capconSpeedNoise
      Message = {$CapconAlarms/MaxSpeed}
      Code = 603
      Severity = 50
    [41]:
      Name = notEnoughFreeMem
      Message = {$dataAlarms/notEnoughFreeMem}
      Code = 604
      Severity = 1000
    [42]:
      Name = cantEmptyNeedCassette
      Message = {$MainAlarms/cantEmptyNeedCassette}
      Code = 605
      Severity = 1000
    [43]:
      Name = opcuaMethodError
      Message = {$MainAlarms/opcuaMethodError}
      Code = 606
      Severity = 1000
    [44]:
      Name = stepperWUError
      Message = {$WingAlarms/StepperWUError}
      Code = 607
  mapp.AlarmX.Core.Snippets:
    [0]:
      Key = linearFeederFaultText
      Value:
        PV = ::vibrator:local_no_opcua[1].axisAlarmText
    [1]:
      Key = circularFeederFaultText
      Value:
        PV = ::vibrator:local_no_opcua[0].axisAlarmText
    [2]:
      Key = beltAxisFaultText
      Value:
        PV = ::belt:this.axisAlarmText
```

### mp_config.mprecipexml - X20CP0484/mappServices/mp_config.mprecipexml
```
Element mpConfig (Type=mprecipexml)
  Alarms = MpAlarmX
    mapp.AlarmX.Core.Configuration:
      [0]:
        Message = {$IAT/SaveFailed}
        Severity = 1000
      [1]:
        Message = {$IAT/SaveFailedPartial}
        Severity = 1000
      [2]:
        Message = {$IAT/LoadFailed}
        Severity = 1000
      [3]:
        Message = {$IAT/LoadFailedPartial}
        Severity = 1000
```

### mp_data.mpdatarecorder - X20CP0484/mappServices/mp_data.mpdatarecorder
```
Element mpData (Type=mpdatarecorder)
  DataRecorder:
    MaxNumberOfFiles = 2
    MaxFileSize = 50000
    BufferSize = 5000
    PowerFailSafe = FALSE
    DecimalMark = .
    AutoSave = FALSE
    OverwriteOldestFile = TRUE
  Alarms = MpAlarmX
    mapp.AlarmX.Core.Configuration:
      [0]:
        Severity = 1000
      [1]:
        Severity = 1000
      [2]:
        Severity = 1000
```

### mp_recipe.mprecipexml - X20CP0484/mappServices/mp_recipe.mprecipexml
```
Element mpRecipe (Type=mprecipexml)
  Alarms = MpAlarmX
    mapp.AlarmX.Core.Configuration:
      [0]:
        Message = {$IAT/SaveFailed}
        Severity = 1000
      [1]:
        Message = {$IAT/SaveFailedPartial}
        Severity = 1000
      [2]:
        Message = {$IAT/LoadFailed}
        Severity = 1000
      [3]:
        Message = {$IAT/LoadFailedPartial}
        Severity = 1000
```

### mp_recipeC.mprecipexml - X20CP0484/mappServices/mp_recipeC.mprecipexml
```
Element mpRecipeCurrent (Type=mprecipexml)
```

### mp_report.mpreportcore - X20CP0484/mappServices/mp_report.mpreportcore
```
Element mpReport (Type=mpreportcore)
  MpReport:
    Settings:
      ResourceDeviceName = IMAGES
      LanguageDependent:
        [0]:
          Language = en
          Font = 1
          DateTimePattern = %Y-%m-%d
    PageLayouts:
      [0]:
        Name = cm20Protocol
        Margins = 2
      [1]:
        Name = cm20Checklist
        Margins = 2
      [2]:
        Name = cm20hwReport
        Margins = 2
    Styles:
      Text:
        [0]:
          Name = Default
          Size = 12
          NumberOfDecimalPlaces = 2
        [1]:
          Name = HeaderText
          Style = 1
          Size = 18
          NumberOfDecimalPlaces = 2
        [2]:
          Name = defaultBold
          Style = 1
          Size = 12
          NumberOfDecimalPlaces = 2
        [3]:
          Name = Default10
          NumberOfDecimalPlaces = 2
        [4]:
          Name = headerChecklist
          Style = 1
          Size = 14
        [5]:
          Name = defaultItalic
          Style = 2
          Size = 12
        [6]:
          Name = default3Decimals
          Size = 12
          NumberOfDecimalPlaces = 3
      Table:
        [0]:
          Name = mainTable
          Padding = 2
      Line:
        [0]:
          Name = horizontalLine
          Width = 3
          Color = 0000FF
      Chart:
        PieChart:
          [0]:
            Name = Default
        LineChart:
          [0]:
            Name = Default
        BarChart:
          [0]:
            Name = Default
    Tables:
      [0]:
        Name = TableContent
        TableStyle = mainTable
        TextStyle = defaultBold
        [0]:
          [0] = TextId
            Source = Type no.- Seial no.:
            Width = 30
          [1] = ValueId
            Value:
              ProcessVariable = ::FAT:resultFAT.additionalInfo.typeNoAndSerialNo
            Width = 30
            HorizontalAlign = 1
          [2] = TextId
            Source = Date:
            Width = 10
            HorizontalAlign = 2
          [3] = DateTime
            Width = 30
            HorizontalAlign = 1
        [1]:
          [0] = TextId
            Source = Machine model:
            Width = 30
            HorizontalAlign = 2
          [1] = ValueId
            Value:
              ProcessVariable = ::FAT:resultFAT.machineSetup.strCfSize
            Width = 30
            HorizontalAlign = 1
          [2] = TextId
            Source = Machine type:
            Width = 10
            HorizontalAlign = 2
          [3] = ValueId
            Value:
              ProcessVariable = ::FAT:resultFAT.machineSetup.strMachineType
            Width = 30
            HorizontalAlign = 1
      [1]:
        Name = vibSpringAdjustTable
        TableStyle = mainTable
        TextStyle = Default
        [0]:
          [0] = TextId
            Source = Spring thickn. (mm)
            Width = 20
            HorizontalAlign = 1
          [1] = TextId
            Source = AMOUNT CF
            Width = 40
            HorizontalAlign = 1
          [2] = TextId
            Source = AMOUNT LF
            Width = 40
            HorizontalAlign = 1
        [1]:
          [0] = TextId
            Source = Spring packet:
            Width = 20
          [1] = TextId
            Source = 1
            Width = 14
            HorizontalAlign = 1
          [2] = TextId
            Source = 2
            Width = 13
            HorizontalAlign = 1
          [3] = TextId
            Source = 3
            Width = 13
            HorizontalAlign = 1
          [4] = TextId
            Source = Belt
            Width = 20
            HorizontalAlign = 1
          [5] = TextId
            Source = CF
            Width = 20
            HorizontalAlign = 1
        [2]  // empty row
          [0] = TextId
            Source =                  
            Width = 20
          [1]:
            Width = 14
          [2]:
            Width = 13
          [3]:
            Width = 13
          [4]:
            Width = 20
          [5]:
            Width = 20
        [3]:
          [0] = TextId
            Source = 0.8 mm
            Width = 20
            HorizontalAlign = 1
          [1] = ValueId
            Value:
              ProcessVariable = ::FAT:resultFAT.CFSpringAdjust.plate08mm[0]
            Width = 14
            HorizontalAlign = 1
          [2] = ValueId
            Value:
              ProcessVariable = ::FAT:resultFAT.CFSpringAdjust.plate08mm[1]
            Width = 13
            HorizontalAlign = 1
          [3] = ValueId
            Value:
              ProcessVariable = ::FAT:resultFAT.CFSpringAdjust.plate08mm[2]
            Width = 13
            HorizontalAlign = 1
          [4] = ValueId
            Value:
              ProcessVariable = ::FAT:resultFAT.LFSpringAdjust.plate08mm[0]
            Width = 20
            HorizontalAlign = 1
          [5] = ValueId
            Value:
              ProcessVariable = ::FAT:resultFAT.LFSpringAdjust.plate08mm[1]
            Width = 20
            HorizontalAlign = 1
        [4]:
          [0] = TextId
            Source = 0.9 mm
            Width = 20
            HorizontalAlign = 1
          [1] = ValueId
            Value:
              ProcessVariable = ::FAT:resultFAT.CFSpringAdjust.plate09mm[0]
            Width = 14
            HorizontalAlign = 1
          [2] = ValueId
            Value:
              ProcessVariable = ::FAT:resultFAT.CFSpringAdjust.plate09mm[1]
            Width = 13
            HorizontalAlign = 1
          [3] = ValueId
            Value:
              ProcessVariable = ::FAT:resultFAT.CFSpringAdjust.plate09mm[2]
            Width = 13
            HorizontalAlign = 1
          [4] = ValueId
            Value:
              ProcessVariable = ::FAT:resultFAT.LFSpringAdjust.plate09mm[0]
            Width = 20
            HorizontalAlign = 1
          [5] = ValueId
            Value:
              ProcessVariable = ::FAT:resultFAT.LFSpringAdjust.plate09mm[1]
            Width = 20
            HorizontalAlign = 1
        [5]:
          [0] = TextId
            Source = 1.5 mm
            Width = 20
            HorizontalAlign = 1
          [1] = ValueId
            Value:
              ProcessVariable = ::FAT:resultFAT.CFSpringAdjust.plate15mm[0]
            Width = 14
            HorizontalAlign = 1
          [2] = ValueId
            Value:
              ProcessVariable = ::FAT:resultFAT.CFSpringAdjust.plate15mm[1]
            Width = 13
            HorizontalAlign = 1
          [3] = ValueId
            Value:
              ProcessVariable = ::FAT:resultFAT.CFSpringAdjust.plate15mm[2]
            Width = 13
            HorizontalAlign = 1
          [4] = ValueId
            Value:
              ProcessVariable = ::FAT:resultFAT.LFSpringAdjust.plate15mm[0]
            Width = 20
            HorizontalAlign = 1
          [5] = ValueId
            Value:
              ProcessVariable = ::FAT:resultFAT.LFSpringAdjust.plate15mm[1]
            Width = 20
            HorizontalAlign = 1
        [6]:
          [0] = TextId
            Source = 2.0 mm
            Width = 20
            HorizontalAlign = 1
          [1] = ValueId
            Value:
              ProcessVariable = ::FAT:resultFAT.CFSpringAdjust.plate20mm[0]
            Width = 14
            HorizontalAlign = 1
          [2] = ValueId
            Value:
              ProcessVariable = ::FAT:resultFAT.CFSpringAdjust.plate20mm[1]
            Width = 13
            HorizontalAlign = 1
          [3] = ValueId
            Value:
              ProcessVariable = ::FAT:resultFAT.CFSpringAdjust.plate20mm[2]
            Width = 13
            HorizontalAlign = 1
          [4] = ValueId
            Value:
              ProcessVariable = ::FAT:resultFAT.LFSpringAdjust.plate20mm[0]
            Width = 20
            HorizontalAlign = 1
          [5] = ValueId
            Value:
              ProcessVariable = ::FAT:resultFAT.LFSpringAdjust.plate20mm[1]
            Width = 20
            HorizontalAlign = 1
        [7]:
          [0] = TextId
            Source = 2.5 mm
            Width = 20
            HorizontalAlign = 1
          [1] = ValueId
            Value:
              ProcessVariable = ::FAT:resultFAT.CFSpringAdjust.plate25mm[0]
            Width = 14
            HorizontalAlign = 1
          [2] = ValueId
            Value:
              ProcessVariable = ::FAT:resultFAT.CFSpringAdjust.plate25mm[1]
            Width = 13
            HorizontalAlign = 1
          [3] = ValueId
            Value:
              ProcessVariable = ::FAT:resultFAT.CFSpringAdjust.plate25mm[2]
            Width = 13
            HorizontalAlign = 1
          [4] = ValueId
            Value:
              ProcessVariable = ::FAT:resultFAT.LFSpringAdjust.plate25mm[0]
            Width = 20
            HorizontalAlign = 1
          [5] = ValueId
            Value:
              ProcessVariable = ::FAT:resultFAT.LFSpringAdjust.plate25mm[1]
            Width = 20
            HorizontalAlign = 1
        [8]:
          [0] = TextId
            Source = Magnetic gab (mm)
            Width = 20
            HorizontalAlign = 1
          [1] = ValueId
            Value:
              ProcessVariable = ::FAT:resultFAT.CFCoilAdjust.magneticGap
            Width = 40
            HorizontalAlign = 1
          [2] = ValueId
            Value:
              ProcessVariable = ::FAT:resultFAT.LFCoilAdjust.magneticGap
            Width = 40
            HorizontalAlign = 1
      [2]:
        Name = measFromLinearizationCFTable
        TableStyle = mainTable
        TextStyle = Default
        [0]:
          [0]:
            Width = 20
          [1] = TextId
            Source = Min
            Width = 20
            HorizontalAlign = 1
          [2] = TextId
            Source = Acutal
            Width = 20
            HorizontalAlign = 1
          [3] = TextId
            Source = Max
            Width = 20
            HorizontalAlign = 1
        [1]:
          [0] = TextId
            Source = Current [A]
            Width = 20
            HorizontalAlign = 1
          [1] = ValueId
            Value:
              ProcessVariable = ::VibratorCo:localHmi[0].minCurrent
            Width = 20
            HorizontalAlign = 1
          [2] = ValueId
            Value:
              ProcessVariable = ::FAT:resultFAT.CFCaliWithHabasit.maxCurrent
            Width = 20
            HorizontalAlign = 1
          [3] = ValueId
            Value:
              ProcessVariable = ::VibratorCo:localHmi[0].maxCurrent
            Width = 20
            HorizontalAlign = 1
        [2]:
          [0] = TextId
            Source = Frequency [Hz]
            Width = 20
            HorizontalAlign = 1
          [1] = ValueId
            Value:
              ProcessVariable = ::VibratorCo:localHmi[0].minResonanceFrequency
            Width = 20
            HorizontalAlign = 1
          [2] = ValueId
            Value:
              ProcessVariable = ::FAT:resultFAT.CFCaliWithHabasit.ressFrequency
            Width = 20
            HorizontalAlign = 1
          [3] = ValueId
            Value:
              ProcessVariable = ::VibratorCo:localHmi[0].maxResonanceFrequency
            Width = 20
            HorizontalAlign = 1
      [3]:
        Name = measFromLinearizationLFTable
        TableStyle = mainTable
        TextStyle = Default
        [0]:
          [0]:
            Width = 20
          [1] = TextId
            Source = Min
            Width = 20
            HorizontalAlign = 1
          [2] = TextId
            Source = Actual
            Width = 20
            HorizontalAlign = 1
          [3] = TextId
            Source = Max
            Width = 20
            HorizontalAlign = 1
        [1]:
          [0] = TextId
            Source = Current [A]
            Width = 20
            HorizontalAlign = 1
          [1] = ValueId
            Value:
              ProcessVariable = ::VibratorCo:localHmi[1].minCurrent
            Width = 20
            HorizontalAlign = 1
          [2] = ValueId
            Value:
              ProcessVariable = ::FAT:resultFAT.LFSpringAdjust.maxCurrent
            Width = 20
            HorizontalAlign = 1
          [3] = ValueId
            Value:
              ProcessVariable = ::VibratorCo:localHmi[1].maxCurrent
            Width = 20
            HorizontalAlign = 1
        [2]:
          [0] = TextId
            Source = Frequency [Hz]
            Width = 20
            HorizontalAlign = 1
          [1] = ValueId
            Value:
              ProcessVariable = ::VibratorCo:localHmi[1].minResonanceFrequency
            Width = 20
            HorizontalAlign = 1
          [2] = ValueId
            Value:
              ProcessVariable = ::FAT:resultFAT.LFSpringAdjust.ressFrequency
            Width = 20
            HorizontalAlign = 1
          [3] = ValueId
            Value:
              ProcessVariable = ::VibratorCo:localHmi[1].maxResonanceFrequency
            Width = 20
            HorizontalAlign = 1
      [4]:
        Name = additionalInformationTable
        TableStyle = mainTable
        TextStyle = Default
        [0]:
          [0] = TextId
            Source = Type no. - Serial no.
            Width = 50
            HorizontalAlign = 1
          [1] = ValueId
            Value:
              ProcessVariable = ::FAT:resultFAT.additionalInfo.typeNoAndSerialNo
            Width = 50
            HorizontalAlign = 1
        [1]:
          [0] = TextId
            Source = Software version:
            Width = 50
            HorizontalAlign = 1
          [1] = ValueId
            Value:
              ProcessVariable = ::machine:this.hmi.version
            Width = 50
            HorizontalAlign = 1
        [2]:
          [0] = TextId
            Source = Vibrator unit type:
            Width = 50
            HorizontalAlign = 1
          [1] = ValueId
            Value:
              ProcessVariable = ::FAT:resultFAT.additionalInfo.vibratorUnitType
            Width = 50
            HorizontalAlign = 1
        [3]:
          [0] = TextId
            Source = Top unit type:
            Width = 50
            HorizontalAlign = 1
          [1] = ValueId
            Value:
              ProcessVariable = ::FAT:resultFAT.additionalInfo.topUnitType
            Width = 50
            HorizontalAlign = 1
        [4]:
          [0] = TextId
            Source = Machine model:
            HorizontalAlign = 1
          [1] = ValueId
            Value:
              ProcessVariable = ::FAT:resultFAT.machineSetup.strCfSize
            HorizontalAlign = 1
          [2] = TextId
            Source = Top serial number:
            HorizontalAlign = 1
          [3] = ValueId
            Value:
              ProcessVariable = ::FAT:resultFAT.additionalInfo.topSerialNo
            HorizontalAlign = 1
        [5]:
          [0] = TextId
            Source = Weigth CF:
            HorizontalAlign = 1
          [1] = ValueId
            Value:
              ProcessVariable = ::FAT:resultFAT.additionalInfo.weightOfCf
            HorizontalAlign = 1
          [2] = TextId
            Source = Voltage:
            HorizontalAlign = 1
          [3] = TextId
            Source = 120V60Hz / 230V50Hz
            HorizontalAlign = 1
        [6]:
          [0] = TextId
            Source = Bolt torque:
            HorizontalAlign = 1
          [1] = TextId
            Source = 100 Nm
            HorizontalAlign = 1
          [2] = TextId
            Source = Cover Habasit MAB 8 E
            Width = 50
            HorizontalAlign = 1
        [7]:
          [0] = TextId
            Source = IRTH Serial NO.:
            Width = 50
            HorizontalAlign = 1
          [1] = ValueId
            Value:
              ProcessVariable = ::FAT:resultFAT.additionalInfo.IRTHno
            Width = 50
            HorizontalAlign = 1
        [8]:
          [0] = TextId
            Source = RNA Product NO.:
            Width = 50
            HorizontalAlign = 1
          [1] = ValueId
            Value:
              ProcessVariable = ::FAT:resultFAT.additionalInfo.rnaProductNo
            Width = 50
            HorizontalAlign = 1
        [9]:
          [0] = ImageId
            Image = leftMachine.jpg
            Width = 50
            HorizontalAlign = 1
          [1] = ImageId
            Image = rightMachine.jpg
            Width = 50
            HorizontalAlign = 1
        [10]:
          [0] = ValueId
            Value:
              ProcessVariable = ::FAT:resultFAT.machineSetup.strIsItALeftMachine
            Width = 50
            HorizontalAlign = 1
          [1] = ValueId
            Value:
              ProcessVariable = ::FAT:resultFAT.machineSetup.strIsItARightMachine
            Width = 50
            HorizontalAlign = 1
      [5]:
        Name = checkListFirstInfo
        TableStyle = mainTable
        TextStyle = Default
        [0]:
          [0] = TextId
            Source = Serienr:
            Width = 20
            HorizontalAlign = 1
          [1] = ValueId
            Value:
              ProcessVariable = ::FAT:resultFAT.additionalInfo.typeNoAndSerialNo
            Width = 30
            HorizontalAlign = 1
          [2] = TextId
            Source = Type:
            Width = 20
            HorizontalAlign = 1
          [3] = TextId
            Source = CM20
            Width = 30
            HorizontalAlign = 1
        [1]:
          [0] = TextId
            Source = Model:
            Width = 20
            HorizontalAlign = 1
          [1] = ValueId
            Value:
              ProcessVariable = ::FAT:resultFAT.machineSetup.strCfSize
            Width = 30
            HorizontalAlign = 1
          [2] = TextId
            Source = Voltage:
            Width = 20
            HorizontalAlign = 1
          [3] = TextId
            Source = 120V/230V
            Width = 30
            HorizontalAlign = 1
        [2]:
          [0] = TextId
            Source = Top unit no:
            Width = 20
            HorizontalAlign = 1
          [1] = ValueId
            Value:
              ProcessVariable = ::FAT:resultFAT.additionalInfo.topUnitType
            Width = 30
            HorizontalAlign = 1
          [2] = TextId
            Source = RNA Product no:
            Width = 20
            HorizontalAlign = 1
          [3] = ValueId
            Value:
              ProcessVariable = ::FAT:resultFAT.additionalInfo.rnaProductNo
            Width = 30
            HorizontalAlign = 1
        [3]:
          [0] = TextId
            Source = IRTH no:
            Width = 20
            HorizontalAlign = 1
          [1] = ValueId
            Value:
              ProcessVariable = ::FAT:resultFAT.additionalInfo.IRTHno
            Width = 30
            HorizontalAlign = 1
          [2] = TextId
            Source = Software version:
            Width = 20
            HorizontalAlign = 1
          [3] = ValueId
            Value:
              ProcessVariable = ::machine:this.hmi.version
            Width = 30
            HorizontalAlign = 1
      [6]:
        Name = visualInspection
        TableStyle = mainTable
        TextStyle = Default
        [0]:
          [0] = TextId
            Source = Ground top inside
            Width = 40
            HorizontalAlign = 1
          [1] = TextId
            Source = X
            Width = 10
            HorizontalAlign = 1
          [2] = TextId
            Source = PE2 (CF scraber)
            Width = 40
            HorizontalAlign = 1
          [3] = TextId
            Source = X
            Width = 10
            HorizontalAlign = 1
        [1]:
          [0] = TextId
            Source = PE3 (On LF)
            Width = 40
            HorizontalAlign = 1
          [1] = TextId
            Source = X
            Width = 10
            HorizontalAlign = 1
          [2] = TextId
            Source = PE4 (On Belt)
            Width = 40
            HorizontalAlign = 1
          [3] = TextId
            Source = X
            Width = 10
            HorizontalAlign = 1
        [2]:
          [0] = TextId
            Source = No step sticker
            Width = 40
            HorizontalAlign = 1
          [1] = TextId
            Source = X
            Width = 10
            HorizontalAlign = 1
          [2] = TextId
            Source = Pacemaker (on CF)
            Width = 40
            HorizontalAlign = 1
          [3] = TextId
            Source = X
            Width = 10
            HorizontalAlign = 1
        [3]:
          [0] = TextId
            Source = Type plate on CF
            Width = 40
            HorizontalAlign = 1
          [1] = TextId
            Source = X
            Width = 10
            HorizontalAlign = 1
          [2] = TextId
            Source = Ground LF
            Width = 40
            HorizontalAlign = 1
          [3] = TextId
            Source = X
            Width = 10
            HorizontalAlign = 1
        [4]:
          [0] = TextId
            Source = Ground top plate
            Width = 40
            HorizontalAlign = 1
          [1] = TextId
            Source = X
            Width = 10
            HorizontalAlign = 1
          [2] = TextId
            Source = Ground bottom inside
            Width = 40
            HorizontalAlign = 1
          [3] = TextId
            Source = X
            Width = 10
            HorizontalAlign = 1
      [7]:
        Name = resistanceMeas1Table
        TableStyle = mainTable
        TextStyle = default3Decimals
        [0]:
          [0] = TextId
            Source = Measuring point
            Width = 30
            HorizontalAlign = 1
          [1] = TextId
            Source = Max. resistance [ohm]
            Width = 30
            HorizontalAlign = 1
          [2] = TextId
            Source = Measured resistance [ohm]
            Width = 40
            HorizontalAlign = 1
        [1]:
          [0] = TextId
            Source = Screw at HMI (PE1)
            Width = 30
            HorizontalAlign = 1
          [1] = TextId
            Source = 0.10
            Width = 30
            HorizontalAlign = 1
          [2] = ValueId
            Value:
              ProcessVariable = ::FAT:resultFAT.resistanceMeas2.measurementArr[0]
            Width = 40
            HorizontalAlign = 1
        [2]:
          [0] = TextId
            Source = Harting, W22
            Width = 30
            HorizontalAlign = 1
          [1] = TextId
            Source = 0.33
            Width = 30
            HorizontalAlign = 1
          [2] = ValueId
            Value:
              ProcessVariable = ::FAT:resultFAT.resistanceMeas2.measurementArr[1]
            Width = 40
            HorizontalAlign = 1
        [3]:
          [0] = TextId
            Source = CF Scraber
            Width = 30
            HorizontalAlign = 1
          [1] = TextId
            Source = 0.10
            Width = 30
            HorizontalAlign = 1
          [2] = ValueId
            Value:
              ProcessVariable = ::FAT:resultFAT.resistanceMeas2.measurementArr[2]
            Width = 40
            HorizontalAlign = 1
        [4]:
          [0] = TextId
            Source = Linear Feeder
            Width = 30
            HorizontalAlign = 1
          [1] = TextId
            Source = 0.10
            Width = 30
            HorizontalAlign = 1
          [2] = ValueId
            Value:
              ProcessVariable = ::FAT:resultFAT.resistanceMeas2.measurementArr[3]
            Width = 40
            HorizontalAlign = 1
        [5]:
          [0] = TextId
            Source = Belt
            Width = 30
            HorizontalAlign = 1
          [1] = TextId
            Source = 0.10
            Width = 30
            HorizontalAlign = 1
          [2] = ValueId
            Value:
              ProcessVariable = ::FAT:resultFAT.resistanceMeas2.measurementArr[4]
            Width = 40
            HorizontalAlign = 1
        [6]:
          [0] = TextId
            Source = Harting, X03
            Width = 30
            HorizontalAlign = 1
          [1] = TextId
            Source = 0.33
            Width = 30
            HorizontalAlign = 1
          [2] = ValueId
            Value:
              ProcessVariable = ::FAT:resultFAT.resistanceMeas2.measurementArr[5]
            Width = 40
            HorizontalAlign = 1
        [7]:
          [0] = TextId
            Source = Harting, X04
            Width = 30
            HorizontalAlign = 1
          [1] = TextId
            Source = 0.33
            Width = 30
            HorizontalAlign = 1
          [2] = ValueId
            Value:
              ProcessVariable = ::FAT:resultFAT.resistanceMeas2.measurementArr[6]
            Width = 40
            HorizontalAlign = 1
        [8]:
          [0] = TextId
            Source = Harting, W22
            Width = 30
            HorizontalAlign = 1
          [1] = TextId
            Source = 0.33
            Width = 30
            HorizontalAlign = 1
          [2] = ValueId
            Value:
              ProcessVariable = ::FAT:resultFAT.resistanceMeas2.measurementArr[7]
            Width = 40
            HorizontalAlign = 1
        [9]:
          [0] = TextId
            Source = Supply, X09:a5
            Width = 30
            HorizontalAlign = 1
          [1] = TextId
            Source = 0.1
            Width = 30
            HorizontalAlign = 1
          [2] = ValueId
            Value:
              ProcessVariable = ::FAT:resultFAT.resistanceMeas2.measurementArr[8]
            Width = 40
            HorizontalAlign = 1
        [10]:
          [0] = TextId
            Source = Supply, X09:a6
            Width = 30
            HorizontalAlign = 1
          [1] = TextId
            Source = 0.1
            Width = 30
            HorizontalAlign = 1
          [2] = ValueId
            Value:
              ProcessVariable = ::FAT:resultFAT.resistanceMeas2.measurementArr[9]
            Width = 40
            HorizontalAlign = 1
      [8]:
        Name = capconVoltageTable
        TableStyle = mainTable
        TextStyle = Default
        [0]:
          [0] = TextId
            Source = Measuring point
            Width = 30
            HorizontalAlign = 1
          [1] = TextId
            Source = Voltage target [V]
            Width = 30
            HorizontalAlign = 1
          [2] = TextId
            Source = Measured voltage [V]
            Width = 40
            HorizontalAlign = 1
        [1]:
          [0] = TextId
            Source = V1 (marking: T2)
            Width = 30
            HorizontalAlign = 1
          [1] = TextId
            Source = 18.5
            Width = 30
            HorizontalAlign = 1
          [2] = ValueId
            Value:
              ProcessVariable = ::FAT:resultFAT.capconMeasurement.V1
            Width = 40
            HorizontalAlign = 1
        [2]:
          [0] = TextId
            Source = V2 (marking: T3)
            Width = 30
            HorizontalAlign = 1
          [1] = TextId
            Source = 15.8
            Width = 30
            HorizontalAlign = 1
          [2] = ValueId
            Value:
              ProcessVariable = ::FAT:resultFAT.capconMeasurement.V2
            Width = 40
            HorizontalAlign = 1
      [9]:
        Name = ioTestTable
        TableStyle = mainTable
        TextStyle = Default
      [10]:
        Name = photoSensorTable
        TableStyle = mainTable
        TextStyle = Default
        [0]:
          [0] = TextId
            Source = Test
            Width = 10
            HorizontalAlign = 1
          [1] = TextId
            Source = Description
            Width = 80
            HorizontalAlign = 1
          [2] = TextId
            Source = Ok:
            Width = 10
            HorizontalAlign = 1
        [1]:
          [0] = TextId
            Source = 1
            Width = 10
            HorizontalAlign = 1
          [1] = TextId
            Source = Mechanical adjustment - the photosensor should be able to detect a 1mm feeler gauge.
            Width = 80
            HorizontalAlign = 1
          [2] = TextId
            Source = X
            Width = 10
            HorizontalAlign = 1
        [2]:
          [0] = TextId
            Source = 2
            Width = 10
            HorizontalAlign = 1
          [1] = TextId
            Source = Run belt continuously for 12s without activation of the photosensor
            Width = 80
            HorizontalAlign = 1
          [2] = TextId
            Source = X
            Width = 10
            HorizontalAlign = 1
      [11]:
        Name = vibratorFreqWithoutHabasitTable
        TableStyle = mainTable
        TextStyle = Default
        [0]:
          [0] = TextId
            Source = Vibrator
            Width = 20
            HorizontalAlign = 1
          [1] = TextId
            Source = Correct freq interval [Hz]
            Width = 40
            HorizontalAlign = 1
          [2] = TextId
            Source = Actual frequency found[Hz]
            Width = 40
            HorizontalAlign = 1
        [1]:
          [0] = TextId
            Source = CF
            Width = 20
            HorizontalAlign = 1
          [1] = ValueId
            Value:
              ProcessVariable = ::FAT:resultFAT.CFSpringAdjust.strTargetFrequency
            Width = 40
            HorizontalAlign = 1
          [2] = ValueId
            Value:
              ProcessVariable = ::FAT:resultFAT.CFSpringAdjust.freqHertz
            Width = 40
            HorizontalAlign = 1
      [12]:
        Name = linearizationWithHabasitCF
        TableStyle = mainTable
        TextStyle = Default
        [0]:
          [0]:
            Width = 20
          [1] = ValueId
            Value:
              ProcessVariable = ::FAT:resultFAT.machineSetup.strMaxSpecsCF
            Width = 20
            HorizontalAlign = 1
          [2] = TextId
            Source = MIN
            Width = 20
            HorizontalAlign = 1
          [3] = ValueId
            Value:
              ProcessVariable = ::FAT:resultFAT.machineSetup.strLinearizationAccValuesCF
            Width = 40
            HorizontalAlign = 1
        [1]:
          [0] = TextId
            Source = Current [A]
            Width = 20
            HorizontalAlign = 1
          [1] = ValueId
            Value:
              ProcessVariable = ::FAT:resultFAT.CFCaliWithHabasit.current100Percent
            Width = 20
            HorizontalAlign = 1
          [2] = ValueId
            Value:
              ProcessVariable = ::FAT:resultFAT.CFCaliWithHabasit.current10Percent
            Width = 20
            HorizontalAlign = 1
          [3] = TextId
            Source = 10% :
            Width = 20
            HorizontalAlign = 1
          [4] = ValueId
            Value:
              ProcessVariable = ::FAT:resultFAT.CFCaliWithHabasit.accValue10Percent
            Width = 20
            HorizontalAlign = 1
        [2]:
          [0] = TextId
            Source = Voltage [V]
            Width = 20
            HorizontalAlign = 1
          [1] = ValueId
            Value:
              ProcessVariable = ::FAT:resultFAT.CFCaliWithHabasit.voltage100Percent
            Width = 20
            HorizontalAlign = 1
          [2] = ValueId
            Value:
              ProcessVariable = ::FAT:resultFAT.CFCaliWithHabasit.voltage10Percent
            Width = 20
            HorizontalAlign = 1
          [3] = TextId
            Source = 100% :
            Width = 20
            HorizontalAlign = 1
          [4] = ValueId
            Value:
              ProcessVariable = ::FAT:resultFAT.CFCaliWithHabasit.accValue100Percent
            Width = 20
            HorizontalAlign = 1
      [13]:
        Name = linearizationWithHabasitLF
        TableStyle = mainTable
        TextStyle = Default
        [0]:
          [0]:
            Width = 20
          [1] = TextId
            Source = MAX (0.09A/200V)
            Width = 20
            HorizontalAlign = 1
          [2] = TextId
            Source = MIN
            Width = 20
            HorizontalAlign = 1
          [3] = ValueId
            Value:
              ProcessVariable = ::FAT:resultFAT.machineSetup.strLinearizationAccValuesLF
            Width = 40
            HorizontalAlign = 1
        [1]:
          [0] = TextId
            Source = Current [A]
            Width = 20
            HorizontalAlign = 1
          [1] = ValueId
            Value:
              ProcessVariable = ::FAT:resultFAT.LFLinearization.current100Percent
            Width = 20
            HorizontalAlign = 1
          [2] = ValueId
            Value:
              ProcessVariable = ::FAT:resultFAT.LFLinearization.current10Percent
            Width = 20
            HorizontalAlign = 1
          [3] = TextId
            Source = 10% :
            Width = 20
            HorizontalAlign = 1
          [4] = ValueId
            Value:
              ProcessVariable = ::FAT:resultFAT.LFLinearization.accValue10Percent
            Width = 20
            HorizontalAlign = 1
        [2]:
          [0] = TextId
            Source = Voltage [V]
            Width = 20
            HorizontalAlign = 1
          [1] = ValueId
            Value:
              ProcessVariable = ::FAT:resultFAT.LFLinearization.voltage100Percent
            Width = 20
            HorizontalAlign = 1
          [2] = ValueId
            Value:
              ProcessVariable = ::FAT:resultFAT.LFLinearization.voltage10Percent
            Width = 20
            HorizontalAlign = 1
          [3] = TextId
            Source = 100% :
            Width = 20
            HorizontalAlign = 1
          [4] = ValueId
            Value:
              ProcessVariable = ::FAT:resultFAT.LFLinearization.accValue100Percent
            Width = 20
            HorizontalAlign = 1
      [14]:
        Name = longTestTable
        TableStyle = mainTable
        TextStyle = Default
        [0]:
          [0]:
            Width = 20
          [1] = TextId
            Source = Test progress [s]
            Width = 40
            HorizontalAlign = 1
          [2] = TextId
            Source = Time left [h]
            Width = 40
            HorizontalAlign = 1
        [1]:
          [0] = TextId
            Source = Test 1 (88h)
            Width = 20
            HorizontalAlign = 1
          [1] = ValueId
            Value:
              ProcessVariable = ::FAT:this.config.timeElapsed88h
            Width = 40
            HorizontalAlign = 1
          [2] = ValueId
            Value:
              ProcessVariable = ::FAT:this.config.timeLeft88h
            Width = 40
            HorizontalAlign = 1
        [2]:
          [0] = TextId
            Source = Test 2 (12h)
            Width = 20
            HorizontalAlign = 1
          [1] = ValueId
            Value:
              ProcessVariable = ::FAT:this.config.timeElapsed12h
            Width = 40
            HorizontalAlign = 1
          [2] = ValueId
            Value:
              ProcessVariable = ::FAT:this.config.timeLeft12h
            Width = 40
            HorizontalAlign = 1
      [15]:
        Name = vibratorFreqWithHabasitTable
        TableStyle = mainTable
        TextStyle = Default
        [0]:
          [0] = TextId
            Source = Vibrator
            Width = 20
            HorizontalAlign = 1
          [1] = TextId
            Source = Correct freq interval [Hz]
            Width = 40
            HorizontalAlign = 1
          [2] = TextId
            Source = Actual frequency found[Hz]
            Width = 40
            HorizontalAlign = 1
        [1]:
          [0] = TextId
            Source = CF
            Width = 20
            HorizontalAlign = 1
          [1] = ValueId
            Value:
              ProcessVariable = ::FAT:resultFAT.CFSpringAdjust.strTargetFrequency
            Width = 40
            HorizontalAlign = 1
          [2] = ValueId
            Value:
              ProcessVariable = ::FAT:resultFAT.CFCaliWithHabasit.freqHertz
            Width = 40
            HorizontalAlign = 1
        [2]:
          [0] = TextId
            Source = LF
            Width = 20
            HorizontalAlign = 1
          [1] = TextId
            Source = 47.5 - 53.5
            Width = 40
            HorizontalAlign = 1
          [2] = ValueId
            Value:
              ProcessVariable = ::FAT:resultFAT.LFSpringAdjust.freqHertz
            Width = 40
            HorizontalAlign = 1
      [16]:
        Name = hwReportTable
        TableStyle = mainTable
        TextStyle = Default
        [0]:
          [0] = TextId
            Source = #
            Width = 6
            HorizontalAlign = 1
          [1] = TextId
            Source = Module name
            Width = 47
            HorizontalAlign = 1
          [2] = TextId
            Source = Module position
            Width = 47
            HorizontalAlign = 1
        [1]:
          [0] = TextId
            Source = 1
            Width = 6
            HorizontalAlign = 1
          [1] = ValueId
            Value:
              ProcessVariable = ::hwReadout:module_cfg[0].mod_name
            Width = 47
            HorizontalAlign = 1
          [2] = ValueId
            Value:
              ProcessVariable = ::hwReadout:module_cfg[0].mod_adress
            Width = 47
            HorizontalAlign = 1
        [2]:
          [0] = TextId
            Source = 2
            Width = 6
            HorizontalAlign = 1
          [1] = ValueId
            Value:
              ProcessVariable = ::hwReadout:module_cfg[1].mod_name
            Width = 47
            HorizontalAlign = 1
          [2] = ValueId
            Value:
              ProcessVariable = ::hwReadout:module_cfg[1].mod_adress
            Width = 47
            HorizontalAlign = 1
        [3]:
          [0] = TextId
            Source = 3
            Width = 6
            HorizontalAlign = 1
          [1] = ValueId
            Value:
              ProcessVariable = ::hwReadout:module_cfg[2].mod_name
            Width = 47
            HorizontalAlign = 1
          [2] = ValueId
            Value:
              ProcessVariable = ::hwReadout:module_cfg[2].mod_adress
            Width = 47
            HorizontalAlign = 1
        [4]:
          [0] = TextId
            Source = 4
            Width = 6
            HorizontalAlign = 1
          [1] = ValueId
            Value:
              ProcessVariable = ::hwReadout:module_cfg[3].mod_name
            Width = 47
            HorizontalAlign = 1
          [2] = ValueId
            Value:
              ProcessVariable = ::hwReadout:module_cfg[3].mod_adress
            Width = 47
            HorizontalAlign = 1
        [5]:
          [0] = TextId
            Source = 5
            Width = 6
            HorizontalAlign = 1
          [1] = ValueId
            Value:
              ProcessVariable = ::hwReadout:module_cfg[4].mod_name
            Width = 47
            HorizontalAlign = 1
          [2] = ValueId
            Value:
              ProcessVariable = ::hwReadout:module_cfg[4].mod_adress
            Width = 47
            HorizontalAlign = 1
        [6]:
          [0] = TextId
            Source = 6
            Width = 6
            HorizontalAlign = 1
          [1] = ValueId
            Value:
              ProcessVariable = ::hwReadout:module_cfg[5].mod_name
            Width = 47
            HorizontalAlign = 1
          [2] = ValueId
            Value:
              ProcessVariable = ::hwReadout:module_cfg[5].mod_adress
            Width = 47
            HorizontalAlign = 1
        [7]:
          [0] = TextId
            Source = 7
            Width = 6
            HorizontalAlign = 1
          [1] = ValueId
            Value:
              ProcessVariable = ::hwReadout:module_cfg[6].mod_name
            Width = 47
            HorizontalAlign = 1
          [2] = ValueId
            Value:
              ProcessVariable = ::hwReadout:module_cfg[6].mod_adress
            Width = 47
            HorizontalAlign = 1
        [8]:
          [0] = TextId
            Source = 8
            Width = 6
            HorizontalAlign = 1
          [1] = ValueId
            Value:
              ProcessVariable = ::hwReadout:module_cfg[7].mod_name
            Width = 47
            HorizontalAlign = 1
          [2] = ValueId
            Value:
              ProcessVariable = ::hwReadout:module_cfg[7].mod_adress
            Width = 47
            HorizontalAlign = 1
        [9]:
          [0] = TextId
            Source = 9
            Width = 6
            HorizontalAlign = 1
          [1] = ValueId
            Value:
              ProcessVariable = ::hwReadout:module_cfg[8].mod_name
            Width = 47
            HorizontalAlign = 1
          [2] = ValueId
            Value:
              ProcessVariable = ::hwReadout:module_cfg[8].mod_adress
            Width = 47
            HorizontalAlign = 1
        [10]:
          [0] = TextId
            Source = 10
            Width = 6
            HorizontalAlign = 1
          [1] = ValueId
            Value:
              ProcessVariable = ::hwReadout:module_cfg[9].mod_name
            Width = 47
            HorizontalAlign = 1
          [2] = ValueId
            Value:
              ProcessVariable = ::hwReadout:module_cfg[9].mod_adress
            Width = 47
            HorizontalAlign = 1
        [11]:
          [0] = TextId
            Source = 11
            Width = 6
            HorizontalAlign = 1
          [1] = ValueId
            Value:
              ProcessVariable = ::hwReadout:module_cfg[10].mod_name
            Width = 47
            HorizontalAlign = 1
          [2] = ValueId
            Value:
              ProcessVariable = ::hwReadout:module_cfg[10].mod_adress
            Width = 47
            HorizontalAlign = 1
        [12]:
          [0] = TextId
            Source = 12
            Width = 6
            HorizontalAlign = 1
          [1] = ValueId
            Value:
              ProcessVariable = ::hwReadout:module_cfg[11].mod_name
            Width = 47
            HorizontalAlign = 1
          [2] = ValueId
            Value:
              ProcessVariable = ::hwReadout:module_cfg[11].mod_adress
            Width = 47
            HorizontalAlign = 1
        [13]:
          [0] = TextId
            Source = 13
            Width = 6
            HorizontalAlign = 1
          [1] = ValueId
            Value:
              ProcessVariable = ::hwReadout:module_cfg[12].mod_name
            Width = 47
            HorizontalAlign = 1
          [2] = ValueId
            Value:
              ProcessVariable = ::hwReadout:module_cfg[12].mod_adress
            Width = 47
            HorizontalAlign = 1
        [14]:
          [0] = TextId
            Source = 14
            Width = 6
            HorizontalAlign = 1
          [1] = ValueId
            Value:
              ProcessVariable = ::hwReadout:module_cfg[13].mod_name
            Width = 47
            HorizontalAlign = 1
          [2] = ValueId
            Value:
              ProcessVariable = ::hwReadout:module_cfg[13].mod_adress
            Width = 47
            HorizontalAlign = 1
        [15]:
          [0] = TextId
            Source = 15
            Width = 6
            HorizontalAlign = 1
          [1] = ValueId
            Value:
              ProcessVariable = ::hwReadout:module_cfg[14].mod_name
            Width = 47
            HorizontalAlign = 1
          [2] = ValueId
            Value:
              ProcessVariable = ::hwReadout:module_cfg[14].mod_adress
            Width = 47
            HorizontalAlign = 1
        [16]:
          [0] = TextId
            Source = 16
            Width = 6
            HorizontalAlign = 1
          [1] = ValueId
            Value:
              ProcessVariable = ::hwReadout:module_cfg[15].mod_name
            Width = 47
            HorizontalAlign = 1
          [2] = ValueId
            Value:
              ProcessVariable = ::hwReadout:module_cfg[15].mod_adress
            Width = 47
            HorizontalAlign = 1
        [17]:
          [0] = TextId
            Source = 17
            Width = 6
            HorizontalAlign = 1
          [1] = ValueId
            Value:
              ProcessVariable = ::hwReadout:module_cfg[16].mod_name
            Width = 47
            HorizontalAlign = 1
          [2] = ValueId
            Value:
              ProcessVariable = ::hwReadout:module_cfg[16].mod_adress
            Width = 47
            HorizontalAlign = 1
        [18]:
          [0] = TextId
            Source = 18
            Width = 6
            HorizontalAlign = 1
          [1] = ValueId
            Value:
              ProcessVariable = ::hwReadout:module_cfg[17].mod_name
            Width = 47
            HorizontalAlign = 1
          [2] = ValueId
            Value:
              ProcessVariable = ::hwReadout:module_cfg[17].mod_adress
            Width = 47
            HorizontalAlign = 1
        [19]:
          [0] = TextId
            Source = 19
            Width = 6
            HorizontalAlign = 1
          [1] = ValueId
            Value:
              ProcessVariable = ::hwReadout:module_cfg[18].mod_name
            Width = 47
            HorizontalAlign = 1
          [2] = ValueId
            Value:
              ProcessVariable = ::hwReadout:module_cfg[18].mod_adress
            Width = 47
            HorizontalAlign = 1
        [20]:
          [0] = TextId
            Source = 20
            Width = 6
            HorizontalAlign = 1
          [1] = ValueId
            Value:
              ProcessVariable = ::hwReadout:module_cfg[19].mod_name
            Width = 47
            HorizontalAlign = 1
          [2] = ValueId
            Value:
              ProcessVariable = ::hwReadout:module_cfg[19].mod_adress
            Width = 47
            HorizontalAlign = 1
    Contents:
      [0]:
        Name = vibSpringAdjustContent
        [0] = Table
          Table = vibSpringAdjustTable
        [1] = EmptyLine
      [1]:
        Name = linearizationResultContentCF
        [0] = Table
          Table = measFromLinearizationCFTable
        [1] = EmptyLine
      [2]:
        Name = linearizationResultContentLF
        [0] = Table
          Table = measFromLinearizationLFTable
      [3]:
        Name = additionalInformation
        [0] = Table
          Table = additionalInformationTable
        [1] = EmptyLine
      [4]:
        Name = footerContentDate
        [0] = DateTime
          Source = ProcessVariable
            ProcessVariable = ::FAT:this.hmi.date
          HorizontalAlign = 2
          NewLine = FALSE
          TextStyle = Default
      [5]:
        Name = checkListFirstInfoContent
        [0] = Table
          Table = checkListFirstInfo
      [6]:
        Name = visualInspectionContent
        [0] = EmptyLine
        [1]:
          Text = 1. Visual inspection of machine mounting and markup
          NewLine = FALSE
          TextStyle = headerChecklist
        [2] = Table
          Table = visualInspection
      [7]:
        Name = resistanceMeas1Content
        [0] = EmptyLine
        [1]:
          Text = 2. Resistance measurements
          TextStyle = headerChecklist
        [2]:
          Text = All measurements are done between PE-clamp in Harting connector in relation to the specified measuring point.
          TextStyle = defaultItalic
        [3] = Table
          Table = resistanceMeas1Table
      [8]:
        Name = capconVoltageContent
        [0] = EmptyLine
        [1]:
          Text = 3. Capcon PSU voltage measurement
          TextStyle = headerChecklist
        [2] = Table
          Table = capconVoltageTable
      [9]:
        Name = ioTestContent
        [0] = EmptyLine
        [1]:
          Text = 4. I/O test
          TextStyle = headerChecklist
        [2]:
          Text = All input and outputs have been tested on the machine from various manuel and automated tests.
          TextStyle = defaultItalic
      [10]:
        Name = levelSensorContent
        [0] = EmptyLine
        [1]:
          Text = 5. Level sensor setup
          TextStyle = headerChecklist
        [2]:
          Text = Adjustments were done manually by a technician and are approved to work properly.
          TextStyle = defaultItalic
      [11]:
        Name = photoSensorContent
        [0] = EmptyLine
        [1]:
          Text = 6. Photosensor setup
          TextStyle = headerChecklist
        [2] = Table
          Table = photoSensorTable
      [12]:
        Name = vibFreqWithoutHabasitContent
        [0] = EmptyLine
        [1]:
          Text = 7. Vibrator frequency without habasit
          TextStyle = headerChecklist
        [2]:
          Text = The machine will do an automatic sweep to find the resonance frequency. Springs are corrected to match the correct operating frequency.
          TextStyle = defaultItalic
        [3] = Table
          Table = vibratorFreqWithoutHabasitTable
      [13]  // For checklist
        Name = linearizationWithoutHabasitContent
        [0] = EmptyLine
        [1]:
          Text = 8. Linearization without habasit
          TextStyle = headerChecklist
        [2]:
          Text = Linearization result for Circular Feeder
          TextStyle = defaultItalic
        [3] = Table
          Table = measFromLinearizationCFTable  // Without habasit!
      [14]:
        Name = longTestContent
        [0] = EmptyLine
        [1]:
          Text = 9. 100 hour test
          TextStyle = headerChecklist
        [2]:
          Text = Machine will run an total of 100 hours. Test 1 should run 88h without habasit in CF. Test 2 should run 12 hours with habasit.
          TextStyle = defaultItalic
        [3]:
          Text = Below it's possible to see if the test was completed.
          TextStyle = defaultItalic
        [4] = Table
          Table = longTestTable
      [15]  // NOT DONE
        Name = vibFreqWithHabasitContent  // For checklist
        [0] = EmptyLine
        [1]:
          Text = 10. Vibrator frequency with habasit
          TextStyle = headerChecklist
        [2] = Table
          Table = vibratorFreqWithHabasitTable
      [16]:
        Name = linearizationWithHabasitContent
        [0] = EmptyLine
        [1]:
          Text = 11. Linearization with habasit
          TextStyle = headerChecklist
        [2]:
          Text = Linearization result for Circular Feeder
          TextStyle = defaultItalic
        [3] = Table
          Table = linearizationWithHabasitCF
        [4]:
          Text = Linearization result for Linear Feeder
          TextStyle = defaultItalic
        [5] = Table
          Table = linearizationWithHabasitLF
      [17]:
        Name = hwReportContent
        [0] = Table
          Table = hwReportTable
    Reports:
      [0]:
        Name = CM20Protocol
        FileNamePattern = Name.pdf
        PageLayout = cm20Protocol
        Footer = footerContentDate
        [0]:
          Heading:
            Text = Protocol for Counting Machine
            HorizontalAlign = 1
            TextStyle = HeaderText
          [0]:
            Content = additionalInformation
        [1]:
          Heading:
            Text = Vibrator adjustments
            HorizontalAlign = 1
            TextStyle = HeaderText
          [0]:
            Content = vibSpringAdjustContent
        [2]:
          Heading:
            Text = Measurements from linearization CF
            HorizontalAlign = 1
            TextStyle = HeaderText
          [0]:
            Content = linearizationResultContentCF
        [3]:
          Heading:
            Text = Measurements from linearization LF
            HorizontalAlign = 1
            TextStyle = HeaderText
          [0]:
            Content = linearizationResultContentLF
      [1]:
        Name = CM20Checklist
        FileNamePattern = Name.pdf
        PageLayout = cm20Checklist
        Footer = footerContentDate
        [0]:
          Heading:
            Text = Checklist for CM20
            HorizontalAlign = 1
            TextStyle = defaultBold
          [0]:
            Content = checkListFirstInfoContent
        [1]:
          Heading:
            Text = 
            TextStyle = headerChecklist
          [0]:
            Content = visualInspectionContent
        [2]:
          Heading:
            Text = 
            TextStyle = headerChecklist
          [0]:
            Content = resistanceMeas1Content
        [3]:
          [0]:
            Content = capconVoltageContent
        [4]:
          [0]:
            Content = ioTestContent
        [5]:
          [0]:
            Content = levelSensorContent
        [6]:
          [0]:
            Content = photoSensorContent
        [7]:
          [0]:
            Content = longTestContent
        [8]:
          Heading:
            Text = CF Calibration
            TextStyle = HeaderText
          [0]:
            Content = linearizationResultContentCF
        [9]:
          Heading:
            Text = LF Calibration
            TextStyle = HeaderText
          [0]:
            Content = linearizationResultContentLF
      [2]:
        Name = CM20hwReport
        FileNamePattern = Name.pdf
        PageLayout = cm20hwReport
        Footer = footerContentDate
        [0]:
          Heading:
            Text = Hardware list for CM20
            TextStyle = HeaderText
          [0]:
            Content = hwReportContent
```

### mp_result.mprecipexml - X20CP0484/mappServices/mp_result.mprecipexml
```
Element mpResult (Type=mprecipexml)
  Alarms = None
```

### mp_user.mpuserx - X20CP0484/mappServices/mp_user.mpuserx
```
Element UserMgmtX (Type=mpuserx)
  Groups:
    DefGroup#1:
      id = Service
      rights:
        [0] = FullAccess
```

### sampWingHw.vvm - X20CP0484/sampWingHw.vvm
```iecst
VAR_CONFIG
	Cyclic#2.::sampling:this.WingHwTOFs[3].OUT AT %Q.Cyclic#3.::bottomFlap:this.hw.di_neighbourChangeover; (*Insert your comment here...*)
	Cyclic#2.::sampling:this.WingHwTOFs[1].OUT AT %Q.Cyclic#3.::middleFlap:this.hw.di_changeover; (*Insert your comment here...*)
	Cyclic#2.::sampling:this.WingHwTOFs[2].OUT AT %Q.Cyclic#3.::bottomFlap:this.hw.di_changeover; (*Insert your comment here...*)
	Cyclic#2.::sampling:this.WingHwTOFs[0].OUT AT %Q.Cyclic#3.::upperFlap:this.hw.di_changeover; (*Insert your comment here...*)
END_VAR
```

### vibrSinWav.vvm - X20CP0484/vibrSinWav.vvm
```iecst
VAR_CONFIG
	Cyclic#2.::sineWaveGe:acc.actVib AT %Q.Cyclic#3.::vibrator:localVariables[0].hw.actVib; (*Insert your comment here...*)
END_VAR
```

## Configuration config1

CPU X20CP0484, AutomationRuntime H4.93, Build 4.1.2, Safety 0.0, Vc 

### Task classes (Cpu.sw)
```
Cyclic#1 (cycle 800 us, tolerance 0 us):
  vibratorCt <- vibratorCtrl.prg
DataObjects: Acp10sys
NcDataObjects: acp10etxen <- acp10etxen.dob, gAxisVibCi <- gAxisVibCobj.gAxisVibCi.dob, cfCurCtr <- gAxisVibCobj.cfCurCtr.dob, gAxisVibLi <- gAxisVibLobj.gAxisVibLi.dob, lfCurCtr <- gAxisVibLobj.lfCurCtr.dob, gAxisBelta <- gAxisBeltobj.gAxisBelta.dob, gAxisBelti <- gAxisBeltobj.gAxisBelti.dob, lfNew <- gAxisVibLobj.lfNew.dob
Binaries: mvLoader, udbdef, FWRules, TCData, TCLang, OpcUaSrv, arsvcreg, acp10cfg, Acp10map, arconfig, User, iomap, asfw, ashwac, ashwd, sysconf, Role, mp_recipe, mp_recipeC, asiol1, User_1, mp_config, mp_data, alarm_hist, TC, mp_user, mp_alarm
Libraries: Acp10man, Acp10par, NcGlobal, MpRecipe, MpBase, sys_lib, runtime, MpAlarmX, astime, brdkMC, Acp10_MC, AsBrMath, standard, AsBrStr, brsystem, brdkMU, brdkSIM, brdkCSV, brdkPV, legoCM20, legoSTR, DataObj, brdkOPCUA, AsOpcUas, brdkUpdate, ArProject, brdkFile, AsSem, AsIO, AsOpcUac, FileIO, AsIODiag, AsUSB, brdkREST, brdkJSON, brdkSTR, RandomLib, AsHttp, AsARCfg, AsMath, asstring, AsEthIP, MTFilter, MTTypes, MTBasics, MTLookUp, MTData, MpData, MpServer, EasyUaClnt, AsIOLink, AsIOAcc, AsUDP, MpReport, powerlnk, arssl, asieccon, aruser
```
